Yaskawa INFORM job: X2_8B-21B(90,180)_DOD_WZMOC_BOK.JBI

/JOB
//NAME X2_8B-21B(90,180)_DOD_WZMOC_BOK
///FOLDERNAME X2
//POS
///NPOS 1035,1035,1035,44,0,0
///TOOL 0
///POSTYPE PULSE
///PULSE
C00000=-1415,-134459,-133802,-1969,12985,79332
C00001=-87080,-112473,-103627,-41798,51237,70410
C00002=-91681,-107347,-99471,-39221,49165,68848
C00003=-93439,-105106,-97054,-38371,48113,68361
C00004=-93441,-104864,-95967,-38672,47682,68565
C00005=-93504,-104969,-96260,-38564,47753,68495
C00006=-95585,-102642,-95415,-36914,47385,67494
C00007=-93504,-104969,-96260,-38564,47753,68495
C00008=-87147,-112175,-102116,-42180,50619,70689
C00009=-87145,-119394,-106475,-25944,48524,38750
C00010=-91166,-110510,-101811,-22693,48895,36705
C00011=-92650,-107060,-99920,-21494,49065,35962
C00012=-94767,-104655,-99060,-19829,49198,34943
C00013=-94484,-105085,-99259,-20052,49173,35080
C00014=-93721,-102513,-96995,-20598,49294,35408
C00015=-94484,-105085,-99259,-20052,49173,35080
C00016=-89209,-117497,-105909,-24366,48468,37757
C00017=-93166,-113214,-115710,-1969,57926,79332
C00018=-93710,-106990,-108704,-1652,56802,79139
C00019=-93766,-106412,-107148,-1629,56140,79127
C00020=-93768,-106433,-106329,-1638,55626,79135
C00021=-93918,-105383,-106173,-1535,56065,79069
C00022=-94164,-101296,-104676,-1361,57240,78956
C00023=-93895,-105502,-106499,-1547,56205,79076
C00024=-93151,-113316,-114305,-1998,57010,79354
C00025=-81072,-99391,-111155,-4750,63110,78553
C00026=-81984,-95120,-104767,-4287,61328,78293
C00027=-82103,-94682,-103397,-4241,60705,78273
C00028=-82106,-94924,-102383,-4271,59960,78300
C00029=-82089,-94934,-102578,-4276,60076,78302
C00030=-82803,-90374,-100753,-3806,61258,77993
C00031=-82089,-94934,-102578,-4276,60076,78302
C00032=-81057,-100006,-109908,-4804,62030,78604
C00033=-94004,-119945,-107122,49530,42714,48164
C00034=-93972,-116281,-97047,53343,39935,45878
C00035=-92833,-103149,-88492,51302,40218,47068
C00036=-93174,-100930,-87132,51219,40604,47120
C00037=-93174,-100493,-85792,51770,40220,46795
C00038=-93174,-101015,-87399,51095,40684,47186
C00039=-92955,-97894,-86230,50180,41136,47726
C00040=-93303,-100448,-87190,51023,40860,47230
C00041=-98055,-98607,-86499,53149,43882,46024
C00042=-96642,-96320,-85623,51883,43475,46780
C00043=-95342,-96864,-85830,51299,42647,47109
C00044=-97130,-98187,-86063,52744,43317,46271
C00045=-114545,-105110,-100746,39625,57097,48369
C00046=-113947,-102413,-97570,39574,56382,48359
C00047=-113947,-102278,-96691,39772,56015,48196
C00048=-113346,-99976,-96570,39024,56612,48763
C00049=-112899,-98120,-95866,38597,56823,49078
C00050=-114020,-99555,-96940,39169,57262,48705
C00051=-56302,-84822,-83054,-58022,66572,84014
C00052=-58361,-85953,-83540,-57558,65172,83717
C00053=-56302,-84822,-83054,-58022,66572,84014
C00054=-50122,-85714,-86741,-59061,71306,84454
C00055=-54195,-101901,-111197,-24063,62262,77343
C00056=-67243,-111926,-101536,21450,29925,69540
C00057=-66442,-101704,-94400,19916,30532,70304
C00058=-66308,-99858,-92576,19846,30336,70336
C00059=-66311,-99589,-91307,20230,29731,70137
C00060=-66308,-99960,-93112,19687,30597,70418
C00061=-70591,-100617,-92786,25268,31264,67678
C00062=-70591,-100325,-91437,25755,30647,67424
C00063=-68222,-99738,-91214,22742,30105,68906
C00064=-70591,-100606,-92729,25289,31242,67667
C00065=-66097,-110297,-96199,21577,27345,69446
C00066=-65719,-107666,-92844,21562,26575,69447
C00067=-65848,-106528,-92445,21497,26927,69482
C00068=-65365,-110699,-93884,21743,25627,69354
C00069=-67243,-111926,-101536,21450,29925,69540
C00070=-68963,-41843,-96211,-398,96948,-48811
C00071=-76932,-51697,-92360,2602,89609,-51106
C00072=-71886,-45093,-85416,705,88639,-49643
C00073=-71886,-45937,-84760,705,87803,-49648
C00074=-71886,-44632,-85753,705,89084,-49641
C00075=-68776,-90352,-95136,-4313,51281,-47645
C00076=-68803,-86754,-93636,-4241,52203,-47695
C00077=-68762,-92243,-95906,-4353,50785,-47617
C00078=-77446,-64871,-91176,8832,74282,-49527
C00079=-75907,-64612,-91046,8095,74185,-49034
C00080=-78150,-64967,-91224,9168,74335,-49752
C00081=-78150,-57569,-97635,8943,81990,-49191
C00082=-68963,-41843,-96211,-398,96948,-48811
C00083=-67385,-42511,-92598,-992,94393,-48367
C00084=-66773,-44328,-90253,-1220,92024,-48175
C00085=-66900,-44765,-89647,-1171,91425,-48205
C00086=-66773,-43962,-90441,-1221,92327,-48178
C00087=-69817,-49291,-93527,-72,91467,-49038
C00088=-102407,-61387,-79216,48101,75803,-74984
C00089=-99741,-62884,-79905,47237,74215,-74494
C00090=-102407,-61387,-79216,48101,75803,-74984
C00091=-71396,-101707,-96198,105,39560,-49678
C00092=-71544,-99303,-95354,247,40276,-49753
C00093=-71126,-105930,-97636,-165,38275,-49535
C00094=-74447,-120283,-111838,3099,39699,-51260
C00095=-57750,-84762,-113304,-22338,79933,-80646
C00096=-38298,-117376,-123136,-35520,84192,-83183
C00097=-31003,-114098,-105660,-45955,85390,-81321
C00098=-32496,-116782,-107403,-45795,84408,-81579
C00099=-34116,-118987,-108120,-45640,83088,-81742
C00100=-33779,-118873,-108083,-45678,83285,-81673
C00101=-33779,-118389,-106291,-45736,82677,-81394
C00102=-33116,-116007,-107005,-45711,84199,-81779
C00103=-43122,-77390,-91933,-43525,86904,-87571
C00104=-44353,-78017,-92219,-43231,86215,-87819
C00105=-45440,-79271,-92786,-42975,85486,-87990
C00106=-45102,-79332,-92813,-43057,85636,-87902
C00107=-45102,-79709,-91490,-43095,84888,-87585
C00108=-41853,-68825,-87871,-43817,88900,-87868
C00109=-48095,-31712,-66541,-47290,99218,-86920
C00110=-48762,-33638,-67810,-47108,98755,-86994
C00111=-49503,-35735,-69173,-46902,98237,-87073
C00112=-49389,-35416,-68966,-46933,98317,-87062
C00113=-49389,-36060,-68028,-46814,97684,-86756
C00114=-48487,-32850,-67294,-47182,98948,-86964
C00115=-45126,-25671,-76382,-49967,106798,-89554
C00116=-48508,-32956,-85951,-38791,109748,-85822
C00117=-73491,-115415,-129730,-12591,84406,-82629
C00118=-68604,-111632,-124361,34026,103601,-55041
C00119=-52690,-105642,-114364,31889,95098,-51390
C00120=-50963,-109289,-114635,31553,93010,-51314
C00121=-50968,-109442,-114037,31534,92627,-51422
C00122=-50963,-109237,-114816,31559,93129,-51281
C00123=-54701,-101748,-112541,32228,96580,-51739
C00124=-54580,-102143,-110625,32107,95358,-52042
C00125=-52710,-105778,-111943,31798,93771,-51772
C00126=-54580,-102143,-110625,32107,95358,-52042
C00127=-53574,-106836,-112314,31893,93817,-52092
C00128=-52008,-102475,-110737,31756,94333,-51344
C00129=-53574,-106836,-112314,31893,93817,-52092
C00130=-61074,-96775,-114868,33501,102293,-52496
C00131=-149084,-102156,-129577,22032,95315,-42360
C00132=-128569,-114069,-129208,14930,94899,-36248
C00133=-124702,-111484,-125119,14131,93099,-35189
C00134=-123206,-111006,-122572,13804,91571,-34868
C00135=-123205,-111346,-122108,13798,91123,-34918
C00136=-123169,-110975,-122344,13795,91444,-34870
C00137=-122647,-104244,-120003,13724,93323,-34489
C00138=-123169,-110975,-122344,13795,91444,-34870
C00139=-116503,-109521,-121739,12400,90787,-32743
C00140=-113941,-110266,-121994,11839,90202,-31960
C00141=-116503,-109521,-121739,12400,90787,-32743
C00142=-121595,-114825,-128025,13496,92670,-34216
C00143=-123984,-121300,-124584,22039,85383,-28695
C00144=-118596,-113071,-118409,20758,84424,-26972
C00145=-117828,-112575,-117002,20585,83663,-26833
C00146=-117596,-112721,-116348,20543,83158,-26838
C00147=-117643,-112201,-116474,20543,83493,-26797
C00148=-117846,-106122,-114344,20549,85245,-26570
C00149=-117643,-112201,-116474,20543,83493,-26797
C00150=-125192,-113488,-115877,22341,84450,-29296
C00151=-124919,-116220,-115928,22323,83104,-29449
C00152=-122352,-116155,-116251,21738,82647,-28614
C00153=-124919,-116220,-115928,22323,83104,-29449
C00154=-123984,-121300,-124584,22039,85383,-28695
C00155=-86442,-134681,-133724,-19248,79211,-32552
C00156=-86002,-121949,-124889,-19319,80358,-32581
C00157=-85994,-121959,-123892,-19351,79775,-32484
C00158=-85995,-122137,-123177,-19379,79272,-32404
C00159=-85938,-122450,-123568,-19392,79360,-32398
C00160=-86651,-115539,-121342,-19081,81262,-32951
C00161=-85938,-122450,-123568,-19392,79360,-32398
C00162=-130270,-119263,-121891,15868,79169,-48216
C00163=-132135,-133974,-122544,16883,72658,-49767
C00164=-129371,-136174,-123179,16117,71390,-48932
C00165=-132135,-133974,-122544,16883,72658,-49767
C00166=-120611,-122953,-119681,21560,80854,-22535
C00167=-120610,-122943,-118608,21593,80243,-22645
C00168=-120610,-122853,-116921,21650,79318,-22813
C00169=-120610,-122881,-117271,21638,79506,-22779
C00170=-120610,-122878,-117279,21638,79511,-22778
C00171=-120610,-122881,-117271,21638,79506,-22779
C00172=-120610,-122873,-117198,21640,79468,-22785
C00173=-120610,-122853,-117190,21640,79473,-22785
C00174=-120610,-122873,-117198,21640,79468,-22785
C00175=-120611,-122910,-120952,21522,81605,-22399
C00176=-86002,-120340,-127953,-19212,82925,-32989
C00177=-85994,-121959,-123892,-19351,79775,-32484
C00178=-85995,-122137,-123177,-19379,79272,-32404
C00179=-85938,-122450,-123568,-19392,79360,-32398
C00180=-86651,-115539,-121342,-19081,81262,-32951
C00181=-85938,-122450,-123568,-19392,79360,-32398
C00182=-130270,-119263,-121891,15868,79169,-48216
C00183=-132135,-133974,-122544,16883,72658,-49767
C00184=-129371,-136174,-123179,16117,71390,-48932
C00185=-132135,-133974,-122544,16883,72658,-49767
C00186=-120612,-120891,-127143,3106,87300,-4415
C00187=-120611,-122177,-124352,3111,84925,-4474
C00188=-120611,-122645,-122467,3116,83527,-4507
C00189=-120611,-122779,-121606,3119,82929,-4523
C00190=-120611,-122697,-122159,3117,83311,-4513
C00191=-120611,-122692,-122166,3117,83318,-4513
C00192=-120611,-122697,-122159,3117,83311,-4513
C00193=-120611,-121412,-126223,3107,86468,-4436
C00194=-96873,-135896,-136150,20148,98342,-27274
C00195=-53188,-122774,-119059,34227,101931,-42117
C00196=-53187,-122644,-116623,34032,100735,-42492
C00197=-53184,-122447,-115007,33919,99986,-42724
C00198=-53180,-122268,-113886,33849,99484,-42877
C00199=-53186,-122531,-115629,33961,100272,-42636
C00200=-53233,-122033,-113114,32057,113501,-44659
C00201=-53229,-122037,-113108,32057,113495,-44659
C00202=-53233,-122033,-113114,32057,113501,-44659
C00203=-53127,-122157,-112856,34567,84618,-41563
C00204=-53132,-122146,-112848,34568,84621,-41564
C00205=-53127,-122157,-112856,34567,84618,-41563
C00206=-53124,-122720,-116247,34514,86111,-41098
C00207=-61684,-126457,-131749,21672,103686,-55019
C00208=-68676,-133744,-131015,10578,108811,-68614
C00209=-80160,-118182,-130261,-41,125141,-81817
C00210=-80187,-122370,-123619,-70,118933,-81856
C00211=-80183,-122639,-122398,-68,118043,-81854
C00212=-80181,-122756,-121636,-67,117515,-81853
C00213=-80184,-122603,-122588,-68,118179,-81854
C00214=-80182,-122615,-122584,-67,118170,-81853
C00215=-80184,-122603,-122588,-68,118179,-81854
C00216=-80200,-121154,-126606,-75,121396,-81862
C00217=-109164,-117358,-132635,-7350,119146,-48306
C00218=-144183,-119511,-130571,-15498,107286,-7245
C00219=-197934,-122815,-127402,-28006,89082,55776
C00220=-202772,-123889,-124791,-27048,85608,54814
C00221=-204705,-124106,-122314,-26692,83530,54575
C00222=-204705,-124189,-120905,-26732,82711,54762
C00223=-205113,-122699,-120601,-26621,83104,54520
C00224=-208506,-122040,-120392,-25870,82241,53457
C00225=-204510,-125657,-121990,-26775,82699,54838
C00226=-204510,-125393,-124777,-26704,84359,54459
C00227=-217123,-144581,-130617,-26990,80795,43719
C00228=-208514,-157553,-136215,-22784,79668,13108
C00229=-208134,-153606,-128050,-23049,77001,13769
C00230=-209226,-147410,-126429,-22728,78719,13024
C00231=-208514,-151468,-127497,-22936,77598,13510
C00232=-208514,-156517,-134755,-22805,79329,13174
C00233=-197934,-122815,-127402,-28006,89082,55776
C00234=-202772,-123889,-124791,-27048,85608,54814
C00235=-204705,-124106,-122314,-26692,83530,54575
C00236=-204705,-124189,-120905,-26732,82711,54762
C00237=-205113,-122699,-120601,-26621,83104,54520
C00238=-208506,-122040,-120392,-25870,82241,53457
C00239=-204510,-125657,-121990,-26775,82699,54838
C00240=-204510,-125393,-124777,-26704,84359,54459
C00241=-217123,-144581,-130617,-26990,80795,43719
C00242=-217745,-144568,-135920,-20596,85340,27526
C00243=-208514,-151468,-127497,-22936,77598,13510
C00244=-209226,-147410,-126429,-22728,78719,13024
C00245=-208514,-151468,-127497,-22936,77598,13510
C00246=-208514,-156517,-134755,-22805,79329,13174
C00247=-187736,-116553,-120968,-36188,98329,31010
C00248=-144869,-104708,-130913,697,92502,-12445
C00249=-97478,-100538,-119508,25976,122096,-72949
C00250=-94415,-115583,-120723,24602,114867,-73486
C00251=-94145,-116737,-119872,24403,113768,-73630
C00252=-94090,-116915,-118863,24267,113100,-73760
C00253=-94227,-118887,-121662,24392,113788,-73658
C00254=-94618,-126072,-123928,23885,111795,-74261
C00255=-93811,-121058,-122280,24303,112998,-73673
C00256=-123165,-134656,-120887,30393,109989,-65140
C00257=-122877,-135920,-118822,30065,108215,-65520
C00258=-120918,-135771,-118381,30417,107339,-64954
C00259=-122877,-135920,-118822,30065,108215,-65520
C00260=-123434,-129548,-123417,31323,113703,-64157
C00261=-126606,-101457,-128935,16844,101795,-36174
C00262=-152779,-135138,-131563,2515,76140,-19155
C00263=-150820,-122490,-124749,1875,78392,-18455
C00264=-150097,-118368,-121531,1645,78513,-18212
C00265=-150095,-118599,-120646,1648,77850,-18220
C00266=-147666,-112236,-119185,871,80184,-17389
C00267=-146670,-110099,-118456,556,80825,-17059
C00268=-148658,-114325,-119887,1186,79554,-17722
C00269=-87079,-91764,-103818,-42328,107533,9448
C00270=-87027,-91004,-101788,-42122,106912,9740
C00271=-89264,-90509,-101588,-42089,105978,9119
C00272=-87027,-91004,-101788,-42122,106912,9740
C00273=-87391,-90282,-107909,-43186,109836,8282
C00274=-92115,-87061,-118989,-19004,94950,-3823
C00275=-78975,-130870,-123203,19746,71053,-12291
C00276=-74317,-97013,-111518,17407,83606,-9286
C00277=-74211,-95430,-110119,17377,83539,-9259
C00278=-74211,-95892,-109317,17397,82840,-9358
C00279=-75305,-113551,-114600,17838,69768,-10493
C00280=-78326,-111051,-111958,19079,70114,-11550
C00281=-78379,-106110,-110225,18937,71523,-11339
C00282=-78263,-116865,-113913,19272,68408,-11810
C00283=-85880,-113569,-112821,22054,71256,-14152
C00284=-85920,-114580,-110580,22309,69503,-14507
C00285=-82054,-114988,-110714,20879,68380,-13249
C00286=-85920,-114580,-110580,22309,69503,-14507
C00287=-78975,-130870,-123203,19746,67177,-12291
C00288=-159950,-115131,-126913,-23322,109234,64770
C00289=-163413,-124246,-126581,-22686,103792,64589
C00290=-164859,-127477,-125491,-22457,101245,64551
C00291=-164857,-127553,-124648,-22406,100728,64651
C00292=-164862,-127370,-126252,-22506,101730,64457
C00293=-158275,-145382,-129341,-21795,96649,67831
C00294=-159759,-153222,-131425,-21726,93697,67826
C00295=-158275,-145382,-129341,-21795,96649,67831
C00296=-157577,-144643,-126617,-21696,95625,68274
C00297=-160219,-140867,-125578,-21868,96138,67212
C00298=-157577,-144643,-126617,-21696,95625,68274
C00299=-152631,-134238,-128202,-21932,102817,68768
C00300=-146941,-123801,-133763,-3444,102850,52685
C00301=-136178,-116173,-124987,31736,84906,22811
C00302=-134413,-106132,-117362,31242,84680,23412
C00303=-134231,-105594,-115694,31219,83968,23286
C00304=-134230,-105863,-115134,31239,83552,23172
C00305=-134007,-104199,-114803,31151,84035,23389
C00306=-133473,-100630,-113499,30965,84737,23780
C00307=-134315,-106237,-115533,31260,83629,23161
C00308=-136272,-117460,-124003,31807,83855,22481
C00309=-136226,-116324,-125056,31750,84893,22789
C00310=-134474,-106353,-117504,31259,84679,23389
C00311=-134275,-105758,-115681,31235,83904,23252
C00312=-134274,-105987,-115198,31252,83547,23154
C00313=-134027,-104733,-115029,31162,83924,23350
C00314=-133465,-100971,-113658,30966,84667,23763
C00315=-134308,-106598,-115693,31262,83551,23142
C00316=-136269,-117902,-124178,31812,83752,22453
C00317=-139753,-124875,-130430,383,75663,-26245
C00318=-143223,-157944,-133481,-5653,58679,-38405
C00319=-140983,-144085,-126452,-6488,61628,-37698
C00320=-140148,-138933,-122655,-6835,62006,-37402
C00321=-140147,-138616,-121921,-6853,61719,-37384
C00322=-140691,-136506,-121897,-6553,62737,-37651
C00323=-138669,-131542,-120459,-7325,64564,-37004
C00324=-140691,-136506,-121897,-6553,62737,-37651
C00325=-145148,-139028,-124584,-4588,62787,-39337
C00326=-159973,-92454,-110285,14523,90938,-48717
C00327=-158765,-97223,-112137,14224,89465,-48492
C00328=-159973,-92454,-110285,14523,90938,-48717
C00329=-164681,-91509,-114703,15696,94847,-49769
C00330=-142525,-105883,-132766,-7713,103357,-60336
C00331=-90751,-115691,-121566,-36045,104861,-61043
C00332=-92920,-122587,-117773,-35137,99152,-60047
C00333=-93124,-123070,-117553,-35091,98753,-60003
C00334=-93124,-123008,-116878,-35050,98435,-59900
C00335=-93160,-123063,-117190,-35068,98555,-59953
C00336=-95752,-125144,-117838,-34977,96947,-60505
C00337=-93160,-123063,-117190,-35068,98555,-59953
C00338=-92038,-109836,-114685,-38536,89453,-57060
C00339=-86810,-100893,-104585,-47463,92019,-56975
C00340=-88449,-102594,-103600,-47188,90148,-56855
C00341=-88449,-102618,-102426,-47172,89639,-56610
C00342=-88449,-102603,-103366,-47184,90046,-56806
C00343=-85133,-99388,-102162,-47637,92393,-56350
C00344=-85168,-99488,-101153,-47595,91912,-56132
C00345=-86978,-101259,-101820,-47360,90627,-56378
C00346=-84037,-98201,-102123,-47804,93363,-56297
C00347=-108771,-112096,-123986,-16313,85813,-59347
C00348=-109769,-112695,-132242,-3132,99947,-61138
C00349=-127404,-127157,-120795,27540,73197,-60883
C00350=-120526,-123085,-115007,25540,69700,-59025
C00351=-119461,-122312,-114032,25210,69192,-58723
C00352=-119461,-122116,-113003,25293,68708,-58832
C00353=-119461,-122312,-114032,25210,69192,-58723
C00354=-94655,-112249,-115827,-1041,75214,-51009
C00355=-93364,-111129,-115444,-1499,75574,-50577
C00356=-121213,-123445,-114215,25873,69302,-59387
C00357=-127714,-127278,-119628,27738,72603,-61150
C00358=-140848,-129628,-128054,17424,84805,-27418
C00359=-127903,-106251,-120637,17388,91568,-15860
C00360=-124887,-98361,-114445,16717,91208,-14907
C00361=-124614,-94849,-112077,16660,91489,-14780
C00362=-117832,-103976,-115449,15062,87719,-13014
C00363=-118209,-109888,-118953,15141,86934,-13233
C00364=-120968,-118649,-124805,15800,86569,-14208
C00365=-112726,-101228,-128594,1890,90279,15897
C00366=-102865,-105549,-130121,-1361,88970,18873
C00367=-85416,-143080,-122146,-23399,58401,32529
C00368=-89847,-131888,-116792,-20882,59491,30436
C00369=-92125,-126361,-114096,-19602,60042,29398
C00370=-92108,-126361,-114086,-19611,60041,29405
C00371=-94963,-119193,-112807,-13876,65309,25883
C00372=-99230,-109273,-111594,-7832,72910,21884
C00373=-97558,-114678,-114533,-8498,72116,22521
C00374=-94805,-124749,-120489,-9597,70928,23580
C00375=-89899,-115674,-129227,-15589,81503,27304
C00376=-94000,-113154,-130859,1035,116659,-75004
C00377=-93721,-118000,-129934,5060,122177,-74127
C00378=-93715,-120352,-127357,4900,119392,-74256
C00379=-95346,-120435,-125547,4467,118331,-74923
C00380=-87734,-123112,-126247,6115,116903,-72103
C00381=-93725,-120284,-127319,4898,119404,-74259
C00382=-93731,-117931,-129895,5059,122189,-74130
C00383=-92605,-107385,-114202,-42080,118626,-78084
C00384=-94957,-117308,-114744,-40643,113912,-77125
C00385=-96859,-119647,-113709,-40343,111617,-77062
C00386=-96820,-119688,-113698,-40330,111613,-77042
C00387=-92369,-120637,-111842,-39132,112371,-75247
C00388=-87506,-133441,-114197,-38673,106213,-75021
C00389=-90618,-118755,-112828,-39302,114392,-75239
C00390=-88476,-109244,-112462,-40625,118981,-76164
C00391=-73726,-95231,-122050,-23824,117115,-78775
C00392=-68964,-113071,-130294,19412,109419,-80322
C00393=-55630,-112625,-122011,35520,97927,-81697
C00394=-52390,-118820,-120628,34805,93310,-81881
C00395=-47869,-106069,-116317,31727,98681,-78960
C00396=-58944,-112669,-113031,37596,97582,-82877
C00397=-56690,-122472,-119439,35129,92879,-83747
C00398=-59872,-116629,-120975,35716,97415,-83571
C00399=-61517,-148095,-119735,48293,75564,-80066
C00400=-55473,-148057,-116974,48060,71191,-79214
C00401=-53771,-146175,-114985,47935,70110,-78894
C00402=-54494,-144748,-112549,48210,69974,-79344
C00403=-55476,-147094,-115701,48129,70996,-79318
C00404=-61520,-147186,-118480,48348,75358,-80173
C00405=-87978,-108563,-128727,6750,125872,-71649
C00406=-93715,-120352,-127357,4900,119392,-74256
C00407=-94869,-122678,-126412,4545,117687,-74766
C00408=-87426,-125031,-126928,6148,116319,-72021
C00409=-93725,-120284,-127319,4898,119404,-74259
C00410=-93731,-117931,-129895,5059,122189,-74130
C00411=-92605,-107385,-114202,-42080,118626,-78084
C00412=-94957,-117308,-114744,-40643,113912,-77125
C00413=-96631,-121222,-114212,-40163,111336,-76837
C00414=-96582,-121324,-114222,-40145,111323,-76807
C00415=-92276,-122277,-112363,-38961,112002,-75057
C00416=-87192,-135738,-114687,-38435,105658,-74669
C00417=-90618,-118755,-112828,-39302,114392,-75239
C00418=-88476,-109244,-112462,-40625,118981,-76164
C00419=-73726,-95231,-122050,-23824,117115,-78775
C00420=-68964,-113071,-130294,19412,109419,-80322
C00421=-55630,-112625,-122011,35520,97927,-81697
C00422=-52390,-118820,-120628,34805,93310,-81881
C00423=-47557,-106620,-116510,31676,98430,-78912
C00424=-58659,-113116,-113184,37566,97351,-82838
C00425=-56690,-122472,-119439,35129,92879,-83747
C00426=-59872,-116629,-120975,35716,97415,-83571
C00427=-61517,-148095,-119735,48293,75564,-80066
C00428=-55473,-148057,-116974,48060,71191,-79214
C00429=-53043,-147267,-115261,47953,69457,-78858
C00430=-53748,-146178,-113424,48182,69442,-79233
C00431=-55476,-147094,-115701,48129,70996,-79318
C00432=-61520,-147186,-118480,48348,75358,-80173
C00433=-69196,-132761,-125763,48066,87564,-77891
C00434=-67178,-112107,-133350,-9560,121946,-71499
C00435=-53652,-115588,-130730,-10921,119132,-80041
C00436=-53631,-118653,-128170,-10572,116038,-79726
C00437=-49406,-129162,-130962,-9295,109096,-77614
C00438=-56866,-119557,-126808,-10903,114346,-80761
C00439=-54665,-117852,-125979,-10629,114989,-80007
C00440=-57520,-119011,-127190,-3009,114777,-80027
C00441=-59278,-121853,-127991,842,113579,-80159
C00442=-55695,-120300,-124998,1328,112531,-78914
C00443=-53493,-120154,-126714,1639,113579,-78070
C00444=-53512,-117734,-129516,1682,116546,-78033
C00445=-64263,-112177,-127274,18013,116425,-52133
C00446=-53349,-113292,-116223,34708,105130,-41711
C00447=-53347,-113647,-113946,34435,103813,-42137
C00448=-52680,-112871,-112467,34368,103124,-42082
C00449=-58031,-122280,-112065,36284,98076,-45699
C00450=-53343,-113729,-112902,34324,103242,-42318
C00451=-53345,-113489,-115217,34581,104530,-41905
C00452=-83368,-135406,-127982,43757,111124,24122
C00453=-107112,-148704,-121184,48737,110155,73723
C00454=-107085,-142005,-111593,48000,108472,72828
C00455=-107084,-140010,-108705,47787,107957,72557
C00456=-87331,-137626,-115833,38185,104318,80918
C00457=-107143,-152743,-127540,-1092,113262,57657
C00458=-106498,-152435,-127519,-1673,113318,57021
C00459=-107059,-148801,-134211,-1989,119286,56706
C00460=-109333,-147161,-118098,47834,110594,72761
C00461=-109333,-141938,-110765,47268,109335,72096
C00462=-106839,-147244,-109723,47050,105697,71521
C00463=-96955,-158208,-128899,-2670,111185,56030
C00464=-107130,-144670,-115956,-40497,90070,47196
C00465=-107133,-145289,-116877,-40503,90261,47122
C00466=-107139,-146938,-119316,-40521,90762,46927
C00467=-81304,-146505,-131302,-46256,99624,33732
C00468=-42290,-135810,-134986,-6789,56953,-43412
C00469=-53482,-111499,-99357,-5283,31563,-44884
C00470=-53488,-110753,-96932,-5448,30458,-44798
C00471=-53106,-110845,-96482,-5998,30161,-44520
C00472=-53143,-110117,-93832,-6189,28906,-44421
C00473=-53188,-109818,-93168,-6175,28651,-44427
C00474=-53095,-108922,-90553,-6542,27518,-44240
C00475=-53472,-108968,-91791,-5862,28222,-44586
C00476=-53466,-109889,-94290,-5675,29282,-44681
C00477=-93748,-113667,-111432,27227,62688,-41579
C00478=-93751,-113561,-109328,27520,61581,-41869
C00479=-94535,-110348,-107800,27711,62471,-41963
C00480=-94560,-109570,-102150,28499,59749,-42715
C00481=-93743,-112935,-104615,28181,59286,-42489
C00482=-93741,-113330,-106821,27872,60309,-42206
C00483=-53707,-103235,-126817,-3349,90409,-72793
C00484=-53694,-107630,-124107,-3352,86490,-72685
C00485=-53689,-108955,-122884,-3357,85060,-72645
C00486=-53697,-108940,-122873,-3354,85062,-72648
C00487=-53721,-108898,-122839,-3346,85062,-72656
C00488=-53729,-108884,-122827,-3345,85059,-72658
C00489=-53735,-107561,-124050,-3339,86489,-72698
C00490=-53748,-103173,-126762,-3336,90406,-72805
C00491=-44251,-68518,-112793,-6305,100072,-70363
C00492=-80270,30794,-42629,-11133,115571,-76543
C00493=-69737,67118,16632,-42575,112328,-80617
C00494=-69636,63823,22197,-49512,110599,-81416
C00495=-67564,55530,12856,-50142,112647,-81508
C00496=-66424,44944,1253,-49852,108764,-84350
C00497=-65618,29495,-14632,-48008,102670,-88237
C00498=-64581,15750,-27557,-48396,103780,-88326
C00499=-64160,11595,-31362,-48525,104124,-88308
C00500=-61878,-10748,-50140,-48981,105285,-87846
C00501=-62672,195,-41330,-51307,112408,-84907
C00502=-58944,10301,-35991,-52571,115494,-84879
C00503=-69716,-6230,-69222,-29298,97742,-75748
C00504=-102330,-22799,-82036,11222,88832,-73278
C00505=-48313,-118911,-129560,19207,92704,-27073
C00506=-53495,-110604,-121584,20154,93282,-28749
C00507=-53898,-112894,-120750,20179,91787,-29140
C00508=-54091,-109968,-119805,20238,92698,-29053
C00509=-54227,-109896,-119946,20266,92849,-29073
C00510=-54259,-112639,-122766,20278,93161,-29031
C00511=-53522,-108468,-123882,20258,95652,-28360
C00512=-66910,-101677,-117691,1645,82254,17515
C00513=-66905,-103395,-115374,1652,79946,17486
C00514=-66559,-103374,-114061,1536,79140,17588
C00515=-66525,-103141,-114029,1523,79241,17602
C00516=-67620,-103650,-114144,1902,79074,17240
C00517=-69811,-106122,-108316,12679,69437,17327
C00518=-66783,-105788,-110032,11324,70201,18483
C00519=-66785,-105108,-112553,11207,72068,18659
C00520=-34610,-119076,-126707,-31995,89279,47352
C00521=-26693,-119602,-105841,-51320,82883,62074
C00522=-26676,-118953,-103885,-51392,82336,62389
C00523=-26611,-118260,-103653,-51381,82509,62328
C00524=-26639,-116853,-99731,-51529,81413,62927
C00525=-26666,-118021,-101324,-51491,81640,62785
C00526=-26683,-118745,-103309,-51412,82173,62476
C00527=-26741,-121947,-116429,-51038,86269,60171
C00528=-80158,-111738,-121779,-46707,81282,-33331
C00529=-80124,-114295,-114082,-47454,77096,-31277
C00530=-80115,-114367,-110881,-47781,75720,-30584
C00531=-79863,-115197,-109969,-48014,75178,-30182
C00532=-79793,-115451,-110067,-48044,75166,-30141
C00533=-80052,-114603,-110983,-47806,75713,-30548
C00534=-80061,-114542,-114188,-47480,77086,-31241
C00535=-80063,-113108,-120040,-30435,104055,-77976
C00536=-80050,-114212,-116860,-30086,101864,-77373
C00537=-80380,-112077,-114717,-30053,101557,-77419
C00538=-79932,-114590,-112006,-35005,85347,-77215
C00539=-79912,-114566,-112044,-35008,85386,-77219
C00540=-80479,-112475,-109427,-36632,80098,-77307
C00541=-80029,-114714,-111597,-36713,80437,-77233
C00542=-82440,-93132,-104306,-35744,84828,-79668
C00543=-83378,-90315,-100640,-35536,83784,-79702
C00544=-86724,-76310,-94495,-34501,85296,-81493
C00545=-81341,-82881,-101909,-35963,88366,-80388
C00546=-80042,-114535,-115070,-36542,82240,-77847
C00547=-80040,-111621,-122742,-8414,85267,-41918
C00548=-80035,-113457,-119567,-8450,82400,-41723
C00549=-81798,-124774,-120168,-7328,73182,-41674
C00550=-80327,-109577,-118133,2572,87034,-53415
C00551=-79380,-112621,-119090,2349,86031,-53125
C00552=-78889,-114029,-118891,6085,83597,-58153
C00553=-80002,-113603,-119620,10752,83390,-63441
C00554=-80006,-103113,-128729,10775,94202,-62513
C00555=-39776,-103787,-110683,-21075,62663,59255
C00556=-39766,-104399,-107995,-21452,60825,59622
C00557=-41663,-99518,-106576,-17765,63773,58656
C00558=-39441,-104963,-106701,-21848,59898,59942
C00559=-39326,-105104,-106740,-21922,59881,59993
C00560=-39744,-104425,-108009,-21464,60826,59630
C00561=-39754,-103814,-110697,-21087,62664,59263
C00562=-47977,-106691,-119962,-23629,83327,62671
C00563=-66867,-99660,-121232,-22132,99220,62132
C00564=-66851,-102572,-118810,-21937,96446,62653
C00565=-74494,-137000,-128982,-14609,78071,53501
C00566=-72467,-138184,-128020,-15181,77278,54315
C00567=-67516,-140688,-126942,-16493,76361,56201
C00568=-43056,-127353,-114280,-36292,85121,62743
C00569=-66851,-103895,-117201,-21852,94891,62938
C00570=-66868,-101493,-119792,-22004,97521,62449
C00571=-74321,-107832,-126985,11736,80239,61811
C00572=-66584,-114412,-108983,34198,49386,64476
C00573=-66581,-113854,-105403,35147,47795,63826
C00574=-59001,-125725,-103773,32485,32454,61113
C00575=-65790,-113886,-101008,36132,45231,63145
C00576=-65568,-123466,-98279,45853,34675,56822
C00577=-65581,-123771,-97752,46366,34344,56544
C00578=-66567,-113311,-102857,35821,46729,63375
C00579=-66569,-114089,-106515,34851,48256,64025
C00580=-52763,-107501,-118592,5184,62268,61653
C00581=-39766,-104399,-107995,-21452,60825,59622
C00582=-42284,-99628,-106389,-17466,63479,58468
C00583=-39837,-104496,-106407,-21621,59851,59791
C00584=-39825,-104515,-106407,-21630,59842,59799
C00585=-39744,-104425,-108009,-21464,60826,59630
C00586=-39754,-103814,-110697,-21087,62664,59263
C00587=-47977,-106691,-119962,-23629,83327,62671
C00588=-66867,-99660,-121232,-22132,99220,62132
C00589=-66851,-102572,-118810,-21937,96446,62653
C00590=-75086,-136456,-128394,-14464,77886,53317
C00591=-72467,-138185,-128020,-15181,77278,54315
C00592=-67516,-140689,-126942,-16493,76360,56201
C00593=-43574,-128187,-114530,-36250,84680,62675
C00594=-66851,-103895,-117201,-21852,94891,62938
C00595=-66868,-101493,-119792,-22004,97521,62449
C00596=-74321,-107832,-126985,11736,80239,61811
C00597=-66584,-114412,-108983,34198,49386,64476
C00598=-66581,-113854,-105403,35147,47795,63826
C00599=-59470,-125293,-103644,32823,32756,60929
C00600=-65940,-113573,-100903,36174,45372,63123
C00601=-65237,-123018,-98144,45460,34612,57042
C00602=-65306,-123403,-97643,46040,34287,56728
C00603=-66567,-113311,-102857,35821,46729,63375
C00604=-66569,-114089,-106515,34851,48256,64025
C00605=-66614,-114312,-115902,32344,53032,65825
C00606=-26293,-124733,-123676,35115,86081,77095
C00607=-26278,-124914,-120130,35186,84196,76502
C00608=-26550,-125631,-118910,35285,83385,76132
C00609=-26140,-123752,-118256,35186,83681,76394
C00610=-26301,-124893,-120124,35190,84211,76498
C00611=-26317,-124710,-123669,35119,86096,77090
C00612=-26368,-124828,-121889,39154,95960,78120
C00613=-26350,-124746,-118556,38992,94373,77544
C00614=-26342,-124553,-116950,38932,93670,77290
C00615=-26340,-123995,-113991,38847,92461,76851
C00616=-26347,-124286,-115407,38884,93032,77056
C00617=-26365,-124761,-118865,39006,94524,77592
C00618=-26264,-124528,-116402,47920,86072,68134
C00619=-26249,-123768,-112787,47988,84810,67516
C00620=-26243,-123374,-111311,48022,84325,67278
C00621=-26226,-122772,-109280,48074,83674,66962
C00622=-26232,-123227,-110778,48035,84146,67194
C00623=-26247,-124165,-114452,47952,85370,67795
C00624=-82585,-123093,-118421,52491,64599,59558
C00625=-107155,-118824,-102398,58122,50036,52281
C00626=-107155,-117467,-98958,59145,49269,51564
C00627=-96813,-117817,-104188,42223,47347,50994
C00628=-105933,-121077,-109912,10415,42869,62990
C00629=-105953,-121074,-109843,10442,42831,62975
C00630=-107149,-121400,-109798,11502,42801,62375
C00631=-106717,-121349,-105974,7567,38238,71665
C00632=-107169,-120346,-107141,7797,39493,71540
C00633=-108433,-119625,-117514,7930,46308,71537
C00634=-107111,-122100,-111275,39348,45202,56077
C00635=-107109,-117760,-98763,43179,41028,53713
C00636=-106761,-117495,-97713,43363,40478,53604
C00637=-106458,-119074,-102370,12274,36991,61895
C00638=-105683,-116022,-101280,9396,37560,63477
C00639=-85991,-103596,-98751,-25015,50891,70344
C00640=-83847,-106333,-107319,-25140,55050,70229
C00641=-110745,-121766,-106380,43469,44759,53583
C00642=-110745,-121766,-106380,43469,44759,53584
C00643=-120731,-110814,-96413,59684,53172,46713
C00644=-94986,-115649,-101302,-12294,38121,75258
C00645=-110957,-117259,-94521,-45268,37979,76630
C00646=-107127,-114270,-91297,-56630,43098,80056
C00647=-102543,-110504,-99650,-53136,49996,77723
C00648=-93612,-109275,-133010,12113,75674,64968
C00649=-74458,-81913,-116300,25886,107898,47202
C00650=-74285,-84923,-113224,25351,104735,46539
C00651=-74085,-86300,-112083,25142,103399,46313
C00652=-71499,-76504,-108067,25490,106819,45523
C00653=-62961,-60085,-100217,24652,107848,48688
C00654=-60437,-59805,-99888,23461,105440,51393
C00655=-60588,-58283,-100875,23679,106756,51616
C00656=-60637,-54628,-103477,24231,109960,52288
C00657=-76657,-70403,-83915,51355,64349,40407
C00658=-74830,-68241,-74355,53953,55282,38932
C00659=-73110,-62379,-68708,53436,54020,39148
C00660=-73126,-62440,-68450,53549,53912,39057
C00661=-36930,-67607,-75173,-26029,44061,77403
C00662=-80523,-89058,-85253,18218,36719,55154
C00663=-82272,-90569,-85112,18702,34759,56728
C00664=-81508,-95500,-88175,18158,33969,56993
C00665=-81043,-103588,-94156,17854,33413,57140
C00666=-82846,-88179,-88219,41798,48730,43563
C00667=-81818,-81213,-82326,41198,48211,43888
C00668=-79663,-80074,-80946,37957,46333,45127
C00669=-64011,-84834,-85332,4259,39755,58703
C00670=-75846,-87347,-86370,15921,40584,52659
C00671=-47572,-67654,-78731,-37306,60592,66422
C00672=-46339,-68382,-80235,-37741,61555,66618
C00673=-42699,-70655,-83815,-39176,63943,67342
C00674=-43803,-67144,-92021,-36183,69839,64523
C00675=-86906,-70734,-117845,25978,101850,24881
C00676=-194376,-118372,-116958,36622,58194,-75254
C00677=-187943,-106127,-101715,33777,52366,-74665
C00678=-187951,-105693,-98645,34509,50978,-75202
C00679=-187954,-105458,-97394,34809,50440,-75417
C00680=-187960,-105469,-97402,34805,50444,-75420
C00681=-187927,-105629,-98482,19599,46235,-60273
C00682=-187923,-105820,-99644,19403,46817,-60144
C00683=-187914,-106157,-102495,18928,48312,-59826
C00684=-188021,-109107,-91072,54887,40419,-77132
C00685=-188025,-108188,-88773,55807,39869,-77674
C00686=-188027,-107805,-87846,56180,39654,-77892
C00687=-188036,-107761,-87717,56242,39627,-77928
C00688=-188035,-108145,-88644,55869,39841,-77710
C00689=-188030,-109068,-90945,54948,40390,-77168
C00690=-188015,-114130,-110744,41340,72657,-75143
C00691=-188018,-113864,-107763,41683,71368,-75679
C00692=-188019,-113684,-106544,41824,70871,-75888
C00693=-188009,-113674,-106577,41816,70886,-75877
C00694=-188008,-113852,-107795,41674,71383,-75668
C00695=-188005,-114114,-110775,41332,72673,-75132
C00696=-187933,-113872,-110928,18210,58720,-57176
C00697=-187882,-113256,-105308,-719,43762,-42538
C00698=-187896,-112711,-102669,-725,42418,-42533
C00699=-187852,-113170,-101841,-775,41671,-42505
C00700=-187778,-112374,-98354,-1639,37547,-42296
C00701=-187899,-111729,-99017,-1491,38283,-42378
C00702=-187886,-112431,-101600,-1465,39511,-42393
C00703=-192869,-127835,-120494,22551,66263,-53872
C00704=-188079,-122619,-114609,40714,83609,-61664
C00705=-188077,-122103,-112045,40794,82601,-62056
C00706=-188097,-121812,-110726,41966,87288,-59780
C00707=-188097,-121769,-110559,41966,87227,-59806
C00708=-188105,-121282,-108770,41980,86589,-60067
C00709=-188106,-121566,-109755,41972,86936,-59927
C00710=-188110,-122188,-112187,41960,87826,-59570
C00711=-188058,-121965,-125191,40549,88870,-59628
C00712=-104402,-90439,-123637,22599,88102,26907
C00713=-80407,-121901,-119741,18448,66455,46046
C00714=-80400,-121844,-116068,18757,64334,45697
C00715=-80358,-121826,-114599,18875,63477,45568
C00716=-79500,-120626,-114191,18436,63629,45929
C00717=-80475,-121542,-115946,18779,64427,45684
C00718=-80482,-121578,-119613,18469,66554,46034
C00719=-85156,-144709,-129107,-21632,59402,64028
C00720=-93856,-120445,-109825,-39450,57641,70752
C00721=-93847,-119691,-106928,-40019,56559,71233
C00722=-86628,-99816,-98593,-45940,69277,74290
C00723=-86043,-99167,-98859,-45014,69635,74495
C00724=-83318,-93529,-94650,-47165,68336,75996
C00725=-93680,-116508,-100417,-40719,46210,72415
C00726=-93820,-118277,-102341,-40471,46353,72255
C00727=-93828,-119232,-105178,-39715,47322,71755
C00728=-93822,-120125,-107980,-28359,52237,38282
C00729=-93816,-119582,-106091,-28689,51458,38525
C00730=-93813,-119346,-105328,-28822,51152,38622
C00731=-93805,-118409,-102529,-29499,49391,39302
C00732=-93820,-119862,-107056,-29266,59584,40856
C00733=-93823,-120114,-107958,-29147,59957,40747
C00734=-93830,-120670,-110185,-28854,60909,40473
C00735=-63807,-119595,-131717,-32346,77391,31957
C00736=-66677,-121755,-125547,-9668,69981,-32239
C00737=-66675,-122709,-116301,-10101,63887,-31721
C00738=-66675,-122586,-115330,-10147,63360,-31673
C00739=-66678,-122782,-121307,9429,81851,-37654
C00740=-66765,-122962,-121469,9451,81867,-37681
C00741=-66675,-122328,-113778,33290,107246,-42961
C00742=-66675,-122499,-114776,33395,107690,-42822
C00743=-66677,-122795,-117228,33681,108831,-42458
C00744=-67830,-119002,-127241,35733,116022,-40496
C00745=-66677,-118144,-130351,-9432,74728,-32617
C00746=-66675,-122709,-116301,-10101,63887,-31721
C00747=-66675,-122566,-115195,-10154,63288,-31666
C00748=-66598,-122626,-121075,9408,81779,-37632
C00749=-62201,-135318,-124907,8438,77184,-36457
C00750=-72253,-125964,-118680,27296,92025,-49108
C00751=-76379,-123759,-128626,28058,99823,-48794
C00752=-71006,-123079,-126009,31798,108132,-44322
C00753=-66720,-122114,-124411,34847,112827,-41144
C00754=-125074,-112778,-121368,18538,134713,-61704
C00755=-173715,-145384,-131232,-10200,126221,-84589
C00756=-173715,-147046,-136936,-18176,117071,-78230
C00757=-173715,-145384,-131232,-55285,56270,-43989
C00758=-121435,-145384,-131232,-55285,56270,-43989
C00759=-118035,-115309,-97908,-59229,55500,-40903
C00760=-129283,-161545,-102403,-79044,40043,-30541
C00761=-116007,-110364,-98843,-57726,100679,-36272
C00762=-114757,-140924,-107985,-56048,95732,-32110
C00763=-114657,-138777,-101995,-58083,106215,-39512
C00764=-102008,-144788,-123359,-59173,119414,-41279
C00765=-15972,-110889,-128286,-10965,59905,-43045
C00766=-15972,-110889,-128286,-10965,59905,-43045
C00767=-101389,-60822,-75148,6919,68546,-70102
C00768=-115790,69230,64798,-8053,66131,-71909
C00769=-120688,105020,73307,-12402,84846,-73777
C00770=-120868,103639,75593,-12409,82749,-73629
C00771=-120940,103216,76680,-12418,81872,-73566
C00772=-120940,103732,79019,-12450,80724,-73451
C00773=-120940,103216,76680,-12418,81872,-73566
C00774=-120298,112004,89967,-12640,78393,-72988
C00775=-120707,106255,82361,-12511,80017,-73298
C00776=-120298,112004,89967,-12640,78393,-72988
C00777=-120228,112105,88453,-12614,79365,-73063
C00778=-120053,112844,85327,-12571,81642,-73235
C00779=-120830,71540,61874,-4756,55589,-66514
C00780=-120535,76858,72419,-5134,51864,-66212
C00781=-120418,79487,77321,-5314,50212,-66075
C00782=-120418,81305,81326,-5435,48689,-65991
C00783=-120418,79487,77321,-5314,50212,-66075
C00784=-121101,73566,71896,-4942,50464,-66384
C00785=-120640,77942,77238,-5256,49458,-66131
C00786=-121101,73566,71896,-4942,50464,-66384
C00787=-121222,71175,67349,-4775,52021,-66512
C00788=-121527,66226,57370,-4418,55590,-66797
C00789=-120817,46858,51705,6808,46216,-80289
C00790=-120487,52530,62238,7041,42645,-80409
C00791=-120357,55197,66992,7170,41090,-80474
C00792=-120357,57219,71131,7393,39594,-80606
C00793=-120357,55197,66992,7170,41090,-80474
C00794=-121171,51687,64922,7778,40638,-80922
C00795=-120657,55397,69123,7546,39918,-80729
C00796=-121171,51687,64922,7778,40638,-80922
C00797=-121307,49062,60252,7635,42163,-80850
C00798=-121648,43436,49847,7373,45678,-80715
C00799=-109578,66950,51259,-9202,73878,-70224
C00800=-101389,-60822,-75148,6919,68546,-70102
C00801=-96929,-90691,-89138,5080,61517,-23019
C00802=-96929,-90691,-89138,5080,61517,27168
C00803=-133997,38575,-5386,4879,105902,64390
C00804=-134430,35731,-4221,4855,103756,64161
C00805=-134605,34666,-3678,4847,102887,64068
C00806=-134604,34193,-2477,4825,101908,64030
C00807=-134605,34666,-3678,4847,102887,64068
C00808=-133324,38381,1851,4717,101326,64430
C00809=-133984,36157,-436,4773,101627,64224
C00810=-133324,38381,1851,4717,101326,64430
C00811=-132740,42105,45,4739,104308,64739
C00812=-159526,23962,790,32225,80504,55500
C00813=-158922,24925,5721,32299,78113,55050
C00814=-158682,25453,8443,32390,76826,54772
C00815=-158681,25549,9587,32465,76269,54609
C00816=-158682,25408,7790,32348,77149,54866
C00817=-160104,22984,7189,32780,76948,54233
C00818=-159169,24509,8648,32575,76492,54477
C00819=-160104,22984,7189,32780,76948,54233
C00820=-160967,21427,101,32642,80299,54873
C00821=-147551,27169,-6215,28445,81493,60312
C00822=-147017,27605,-1759,28452,79091,59917
C00823=-146805,27803,661,28506,77793,59674
C00824=-146803,27699,1600,28565,77235,59535
C00825=-146805,27874,109,28472,78126,59757
C00826=-148390,24338,-1607,29025,77984,59121
C00827=-147556,26192,183,28786,77573,59333
C00828=-148390,24338,-1607,29025,77984,59121
C00829=-149162,23542,-7999,28991,81344,59682
C00830=-129846,-17397,-52274,16165,101048,68229
C00831=-103949,-6271,-30701,7884,96105,76175
C00832=-94102,16895,-5866,4380,94047,79161
C00833=-94024,14878,-3719,4358,91692,79105
C00834=-93993,14152,-2780,4351,90742,79083
C00835=-93993,14253,-1030,4349,89719,79047
C00836=-93993,14152,-2780,4351,90742,79083
C00837=-93685,20015,4382,4321,89334,79138
C00838=-93881,17120,1686,4338,89515,79078
C00839=-93685,20015,4382,4321,89334,79138
C00840=-93796,22544,1176,4343,92603,79213
C00841=-95224,-25687,-42365,27028,60157,72238
C00842=-94111,-23276,-36997,26973,57954,72128
C00843=-93676,-22245,-34794,26967,57075,72081
C00844=-93677,-22196,-33100,27266,56165,71832
C00845=-93676,-22245,-34794,26967,57075,72081
C00846=-94165,-26445,-35973,27662,55954,71554
C00847=-93910,-23559,-33944,27450,56079,71704
C00848=-94165,-26445,-35973,27662,55954,71554
C00849=-95768,-30118,-43626,27714,58991,71694
C00850=-97625,-41604,-59467,17173,89706,-8843
C00851=-96114,-37688,-53918,16886,88057,-8555
C00852=-95526,-36022,-51615,16777,87400,-8443
C00853=-95527,-36150,-50037,16784,86406,-8579
C00854=-95526,-36022,-51615,16777,87400,-8443
C00855=-95532,-36183,-50637,16782,86745,-8534
C00856=-95234,-33170,-48668,16723,87008,-8396
C00857=-95532,-36183,-50637,16782,86745,-8534
C00858=-95504,-36095,-50208,16778,86530,-8554
C00859=-93996,-36675,-50581,16493,86163,-8084
C00860=-95504,-36095,-50208,16778,86530,-8554
C00861=-97625,-41604,-59467,17173,89706,-8843
C00862=-101873,-77751,-87156,42969,63075,62474
C00863=-95937,-74809,-81328,40948,58735,63434
C00864=-95565,-74583,-80935,40815,58468,63500
C00865=-95566,-74620,-79294,41227,57681,63141
C00866=-95565,-74583,-80935,40815,58468,63500
C00867=-98755,-73227,-80296,42221,60183,62682
C00868=-98803,-73638,-78797,42678,59356,62269
C00869=-96868,-74481,-79195,41849,58298,62761
C00870=-98803,-73638,-78797,42678,59356,62269
C00871=-97163,-69666,-76891,41573,59236,63045
C00872=-96752,-66139,-75134,41097,59602,63417
C00873=-97163,-69666,-76891,41573,59236,63045
C00874=-101873,-77751,-87156,42969,63075,62474
C00875=-126113,-49786,-51573,51544,90004,55144
C00876=-123973,-50127,-48217,51392,87374,54806
C00877=-123286,-49758,-46380,51349,86473,54664
C00878=-118478,-34750,-37348,50925,85086,56432
C00879=-119272,-35479,-39244,50973,86038,56539
C00880=-121232,-35158,-42579,51146,88553,56901
C00881=-111145,-57425,-62081,41633,61582,55088
C00882=-109620,-53993,-56645,41578,59663,54986
C00883=-109014,-52418,-54338,41560,58914,54950
C00884=-105531,-54881,-55720,40219,56972,55856
C00885=-106107,-56401,-57979,40230,57706,55889
C00886=-107578,-60042,-63488,40293,59558,55964
C00887=-93331,-25535,-46307,22677,87971,72102
C00888=-84242,-5399,-27465,11713,100257,81196
C00889=-83743,-8192,-25851,11599,97806,81134
C00890=-83603,-8644,-24372,11558,96668,81075
C00891=-80847,-8673,-24279,11462,96208,81977
C00892=-80973,-8366,-25985,11504,97411,82047
C00893=-81511,-5615,-27635,11617,99868,82095
C00894=-103949,-6271,-30701,7884,96105,76175
C00895=-129846,-17397,-52274,16165,101048,68229
C00896=-175693,57260,35469,48998,74273,48315
C00897=-174652,59964,42108,49342,71909,47593
C00898=-173987,58917,42535,48748,68669,47097
C00899=-173562,58305,42809,47399,62634,46211
C00900=-173482,53917,36869,46602,62532,46609
C00901=-174364,49990,29079,45939,64941,47387
C00902=-163099,39792,11105,47007,80916,54866
C00903=-161954,40669,15666,46993,78691,54338
C00904=-161675,41954,18470,47071,77805,54042
C00905=-160520,35916,12218,46685,77730,54566
C00906=-160850,34862,9687,46632,78611,54832
C00907=-162019,34035,5199,46665,80839,55343
C00908=-147988,42797,109,12455,106225,61454
C00909=-148219,40121,1423,12320,104123,61157
C00910=-148209,38525,1410,12269,103328,61081
C00911=-147238,35306,-1899,12234,103563,61431
C00912=-146513,33084,-4151,12206,103702,61693
C00913=-146794,35355,-3496,12271,104485,61677
C00914=-146567,38090,-4821,12411,106625,61976
C00915=-96929,-90691,-89138,5080,61517,27168
C00916=-96929,-90691,-89138,5080,61517,-23019
C00917=-101389,-60822,-75148,6919,68546,-70102
C00918=-109578,66950,51259,-9202,73878,-70224
C00919=-119285,73548,61078,-7759,54489,-67872
C00920=-119140,78931,71700,-8230,50768,-67516
C00921=-119083,81584,76629,-8462,49121,-67350
C00922=-122917,98444,98202,-6801,44189,-68705
C00923=-122308,90513,86215,-6785,47517,-68668
C00924=-122473,83260,72935,-6271,51921,-69036
C00925=-119074,82203,59752,-14757,75142,-72556
C00926=-112473,77653,55392,-16315,76732,-70397
C00927=-111583,66581,50085,-22599,68947,-68307
C00928=-112205,67748,51306,-22435,68636,-68485
C00929=-112291,70891,55012,-22505,67993,-68392
C00930=-120890,75924,58725,-8799,66214,-71114
C00931=-120891,72538,54662,-8752,66965,-71172
C00932=-121396,73617,55948,-8591,66676,-71337
C00933=-121396,72779,51526,-8459,68942,-71502
C00934=-134157,70152,49704,15847,72235,-43808
C00935=-133722,73949,59265,16087,68355,-44178
C00936=-133862,75249,62165,16247,67307,-44381
C00937=-129675,65866,51066,4701,64817,-31992
C00938=-128682,62362,47014,4314,65455,-31601
C00939=-130205,57581,36634,4742,69462,-32000
C00940=-130312,54578,33992,4779,69550,-32035
C00941=-129992,46081,35923,20239,67004,8502
C00942=-121496,43425,36833,5893,59088,22773
C00943=-120237,47252,43120,2387,56768,25932
C00944=-119972,47626,45454,2298,55515,26011
C00945=-128073,50557,47782,20949,62737,7811
C00946=-127834,53853,52717,21124,61417,7650
C00947=-123180,48310,46556,9691,56439,19302
C00948=-122651,35401,27095,8965,61652,19959
C00949=-109578,66950,51259,-9202,73878,-70224
C00950=-101389,-60822,-75148,6919,68546,-70102
C00951=-96929,-90691,-89138,5080,61517,-23019
C00952=-93242,-109726,-96296,3420,55961,28393
C00953=-92156,-22649,-39625,10516,94476,60392
C00954=-92549,-23820,-36378,10508,91967,60047
C00955=-92689,-24290,-35079,10509,90961,59915
C00956=-95254,-23373,-34430,10727,91365,59075
C00957=-94898,-22950,-35761,10710,92338,59280
C00958=-94492,-21797,-39017,10723,94837,59633
C00959=-92575,-26977,-42679,21088,73618,56030
C00960=-92430,-25186,-37423,21282,71416,55682
C00961=-92290,-24713,-35488,21345,70493,55566
C00962=-95616,-23226,-34216,23502,71566,54461
C00963=-95477,-23933,-36320,23344,72386,54682
C00964=-95719,-25683,-41558,23174,74597,55037
C00965=-96929,-90691,-89138,5080,61517,27168
C00966=-96929,-90691,-89138,5080,61517,-23019
C00967=-101389,-60822,-75148,6919,68546,-70102
C00968=-109578,66950,51259,-9202,73878,-70224
C00969=-108278,48890,46404,-6655,48460,-73563
C00970=-108252,54023,56228,-7048,45078,-73302
C00971=-108672,56895,61153,-6970,43500,-73378
C00972=-113114,65075,70630,-4174,41573,-75428
C00973=-112702,61866,65174,-4315,43297,-75310
C00974=-112766,56024,54314,-4011,46966,-75508
C00975=-103921,32533,46603,10708,30188,-75698
C00976=-104692,35200,60863,30413,16065,-83251
C00977=-104796,38679,66061,33302,14894,-84599
C00978=-102333,36267,63497,27606,14351,-81669
C00979=-100412,37194,55383,7603,26828,-73795
C00980=-100998,29868,43914,7479,30147,-73786
C00981=-109578,66950,51259,-9202,73878,-70224
C00982=-101389,-60822,-75148,6919,68546,-70102
C00983=-96929,-90691,-89138,5080,61517,-23019
C00984=-96929,-90691,-89138,5080,61517,27168
C00985=-90570,-23240,-39845,-1682,91658,61068
C00986=-90349,-1837,-19216,-4288,101242,62233
C00987=-90005,-3734,-19299,-4261,100340,62382
C00988=-92752,-2865,-18588,-4343,100202,61442
C00989=-95291,-22836,-35623,-1093,89189,59526
C00990=-94239,-22001,-38963,-1226,91687,59852
C00991=-90424,-29050,-43505,3763,58999,61302
C00992=-86008,-21130,-36360,-6353,62529,61992
C00993=-86454,-19207,-33152,-6175,61515,61881
C00994=-89453,-18520,-32647,-4592,61359,60761
C00995=-95351,-24457,-36663,6763,57473,59317
C00996=-94707,-27619,-42528,6252,59394,59681
C00997=-109011,-26713,-50438,8452,98222,74634
C00998=-144543,31549,-11380,-159,92982,60584
C00999=-143093,45679,4448,-4866,97184,60249
C01000=-143214,43522,5393,-4827,95492,60276
C01001=-146471,54490,17318,-4285,93619,59288
C01002=-148937,42537,3991,922,89189,59187
C01003=-148250,43318,770,754,91565,59420
C01004=-172279,3947,-14828,46151,77384,48319
C01005=-167570,-10636,-17777,41693,62852,42800
C01006=-166655,-7092,-11488,42082,60867,42363
C01007=-169056,5005,-1455,42887,62060,41693
C01008=-172859,17944,7820,47479,72977,45875
C01009=-174013,15583,1984,47261,75226,46421
C01010=-109011,-26713,-50438,8452,98222,74634
C01011=-99312,-50897,-61026,22837,72179,74454
C01012=-98138,-49989,-56545,22703,69739,74412
C01013=-106382,-52347,-50887,37007,65807,70627
C01014=-98813,-18962,-39289,22939,92751,75811
C01015=-101547,-27333,-44313,25543,91651,74875
C01016=-97857,-18198,-39852,20610,99055,76884
C01017=-96922,-25876,-47272,18742,95048,76352
C01018=-97638,-23312,-49453,18962,97729,76524
C01019=-81141,-50558,-66105,12803,46081,75388
C01020=-80687,-46119,-60183,12697,44679,75401
C01021=-80513,-44339,-57785,12667,44105,75401
C01022=-80516,-44488,-54802,13120,42239,75121
C01023=-80690,-46329,-57233,13145,42803,75122
C01024=-81145,-50923,-63237,13239,44177,75109
C01025=-83601,15534,-39616,9664,96262,77072
C01026=-80484,90945,50155,4324,118905,78550
C01027=-80490,84570,45509,4303,118490,78531
C01028=-80493,82108,43801,4293,118276,78521
C01029=-80495,81630,46278,4216,116511,78452
C01030=-80492,84058,47940,4226,116735,78462
C01031=-83493,53381,-2692,9637,111099,78940
C01032=-91945,-14209,-43630,9790,83010,75128
C01033=-10907,-117335,-90652,-18762,63715,-59495
C01034=-15972,-110889,-128286,-10965,59905,-43045
BC00000=48829,688840,1075175
BC00001=366911,902233,1075175
BC00002=366911,902233,1075175
BC00003=366911,902233,1075175
BC00004=366911,902233,1075175
BC00005=366911,902233,1075175
BC00006=366911,902233,1075175
BC00007=366911,902233,1075175
BC00008=366911,902233,1075175
BC00009=333056,895412,1075175
BC00010=333056,895412,1075175
BC00011=333056,895412,1075175
BC00012=333056,895412,1075175
BC00013=333056,895412,1075175
BC00014=333056,895412,1075175
BC00015=333056,895412,1075175
BC00016=333056,895412,1075175
BC00017=358091,902222,1075175
BC00018=358091,902222,1075175
BC00019=358091,902222,1075175
BC00020=358091,902222,1075175
BC00021=358091,902222,1075175
BC00022=358091,902222,1075175
BC00023=358091,902222,1075175
BC00024=358091,902222,1075175
BC00025=398174,894103,1075175
BC00026=398174,894103,1075175
BC00027=398174,894103,1075175
BC00028=398174,894103,1075175
BC00029=398174,894103,1075175
BC00030=398174,894103,1075175
BC00031=398174,894103,1075175
BC00032=398174,894103,1075175
BC00033=264903,781270,1075175
BC00034=264903,781270,1075175
BC00035=264904,781269,1075172
BC00036=264904,781269,1075171
BC00037=264904,781269,1075171
BC00038=264904,781269,1075168
BC00039=264904,781269,1075168
BC00040=264904,781269,1075168
BC00041=264904,781269,1075168
BC00042=264904,781269,1075168
BC00043=264904,781269,1075164
BC00044=264903,781270,1075175
BC00045=301264,775814,1075175
BC00046=301264,775814,1075175
BC00047=301264,775814,1075175
BC00048=301264,775814,1075175
BC00049=301264,775814,1075175
BC00050=301264,775814,1075175
BC00051=301264,775814,1075175
BC00052=301264,775814,1075175
BC00053=301264,775814,1075175
BC00054=301264,775814,1075175
BC00055=274235,786209,1075175
BC00056=238672,799885,1075175
BC00057=238672,799885,1075175
BC00058=238672,799885,1075175
BC00059=238672,799885,1075175
BC00060=238672,799885,1075175
BC00061=238672,799885,1075175
BC00062=238672,799885,1075175
BC00063=238672,799885,1075175
BC00064=238672,799884,1075171
BC00065=238672,799884,1075171
BC00066=238672,799885,1075175
BC00067=238672,799885,1075175
BC00068=238672,799885,1075175
BC00069=238672,799885,1075175
BC00070=318263,750454,1075175
BC00071=318263,750454,1075175
BC00072=318263,750454,1075175
BC00073=318263,750454,1075175
BC00074=318263,750454,1075175
BC00075=318263,750454,1075175
BC00076=318263,750454,1075175
BC00077=318263,750454,1075175
BC00078=318263,750454,1075175
BC00079=318263,750454,1075175
BC00080=318263,750454,1075175
BC00081=318263,750454,1075175
BC00082=318263,750454,1075175
BC00083=318263,750454,1075175
BC00084=318263,750454,1075175
BC00085=318263,750454,1075175
BC00086=318263,750454,1075175
BC00087=318263,750454,1075175
BC00088=318263,750454,1075175
BC00089=318263,750454,1075175
BC00090=318263,750454,1075175
BC00091=318263,750454,1075175
BC00092=318263,750454,1075175
BC00093=318263,750454,1075175
BC00094=318263,750454,1075175
BC00095=377114,750454,1075175
BC00096=397814,750454,1075175
BC00097=397814,750454,1075175
BC00098=397814,750454,1075175
BC00099=397814,750454,1075175
BC00100=397814,750454,1075175
BC00101=397814,750454,1075175
BC00102=397814,750454,1075175
BC00103=397814,750454,1075175
BC00104=397814,750454,1075175
BC00105=397814,750454,1075175
BC00106=397814,750454,1075175
BC00107=397814,750454,1075175
BC00108=397814,750454,1075175
BC00109=397814,750454,1075175
BC00110=397814,750454,1075175
BC00111=397814,750454,1075175
BC00112=397814,750454,1075175
BC00113=397814,750454,1075175
BC00114=397814,750454,1075175
BC00115=397814,750454,1075175
BC00116=383090,762961,1075175
BC00117=372387,772052,1075175
BC00118=296274,836703,1075175
BC00119=296274,836703,1075175
BC00120=296274,836703,1075175
BC00121=296274,836703,1075175
BC00122=296274,836703,1075175
BC00123=296274,836703,1075175
BC00124=296274,836703,1075175
BC00125=296274,836703,1075175
BC00126=296274,836703,1075175
BC00127=296274,836703,1075175
BC00128=296274,836703,1075175
BC00129=296274,836703,1075175
BC00130=296274,836703,1075175
BC00131=312215,899988,1075175
BC00132=312215,944285,1075175
BC00133=312215,944285,1075175
BC00134=312215,944285,1075175
BC00135=312215,944285,1075175
BC00136=312215,944285,1075175
BC00137=312215,944285,1075175
BC00138=312215,944285,1075175
BC00139=312215,944285,1075175
BC00140=312215,944285,1075175
BC00141=312215,944285,1075175
BC00142=312215,944285,1075175
BC00143=259299,938961,1075175
BC00144=259299,938961,1075175
BC00145=259299,938961,1075175
BC00146=259299,938961,1075175
BC00147=259299,938961,1075175
BC00148=259299,938961,1075175
BC00149=259299,938961,1075175
BC00150=259299,938961,1075175
BC00151=259299,938961,1075175
BC00152=259299,938961,1075175
BC00153=259299,938961,1075175
BC00154=259299,938961,1075175
BC00155=211531,951911,1075175
BC00156=211531,951911,1075175
BC00157=211531,951911,1075175
BC00158=211531,951911,1075175
BC00159=211531,951911,1075175
BC00160=211531,951911,1075175
BC00161=211531,951911,1075175
BC00162=211531,951911,1075175
BC00163=211531,951911,1075175
BC00164=211531,951911,1075175
BC00165=211531,951911,1075175
BC00166=182503,951872,1075175
BC00167=184369,953383,1075175
BC00168=184369,953399,1075175
BC00169=184333,953526,1075175
BC00170=184897,956550,1075175
BC00171=184333,953526,1075175
BC00172=184751,953664,1075175
BC00173=187887,953121,1075175
BC00174=184751,953664,1075175
BC00175=178222,948378,1075175
BC00176=171711,951911,1075175
BC00177=171711,959591,1075175
BC00178=171711,959591,1075175
BC00179=171711,959591,1075175
BC00180=171711,959591,1075175
BC00181=171711,959591,1075175
BC00182=171711,959591,1075175
BC00183=171711,959591,1075175
BC00184=171711,959591,1075175
BC00185=171711,959591,1075175
BC00186=182815,952263,1075175
BC00187=183711,957103,1075175
BC00188=184069,959047,1075174
BC00189=184070,959056,1075175
BC00190=184189,959079,1075175
BC00191=184752,962103,1075175
BC00192=184189,959079,1075175
BC00193=182935,952303,1075175
BC00194=148303,998123,1075175
BC00195=123088,1061215,1075175
BC00196=126332,1055781,1075175
BC00197=127630,1053613,1075175
BC00198=127630,1053623,1075175
BC00199=127630,1053607,1075175
BC00200=153753,1064749,1075175
BC00201=152152,1062093,1075175
BC00202=153753,1064749,1075175
BC00203=104366,1038154,1075175
BC00204=107120,1036610,1075175
BC00205=104366,1038154,1075175
BC00206=97490,1044180,1075175
BC00207=121157,1044973,1075175
BC00208=140343,1045718,1075175
BC00209=158643,1046375,1075175
BC00210=155464,1041036,1075175
BC00211=155106,1040455,1075175
BC00212=155106,1040463,1075175
BC00213=155288,1040367,1075175
BC00214=153687,1037711,1075175
BC00215=155288,1040367,1075175
BC00216=158891,1046297,1075175
BC00217=211337,993614,1075175
BC00218=274623,983932,1075175
BC00219=371761,1043051,1075175
BC00220=331941,1063020,1075175
BC00221=331941,1063020,1075175
BC00222=331941,1063020,1075175
BC00223=331941,1063020,1075175
BC00224=331941,1063020,1075175
BC00225=331941,1063020,1075175
BC00226=331941,1063020,1075175
BC00227=331941,1063020,1075175
BC00228=331941,1063020,1075175
BC00229=331941,1063020,1075175
BC00230=331941,1063020,1075175
BC00231=331941,1063020,1075175
BC00232=331941,1063020,1075175
BC00233=371761,1043051,1075175
BC00234=371761,1043051,1075175
BC00235=371761,1043051,1075175
BC00236=371761,1043051,1075175
BC00237=371761,1043051,1075175
BC00238=371761,1043051,1075175
BC00239=371761,1043051,1075175
BC00240=371761,1043051,1075175
BC00241=371761,1043051,1075175
BC00242=371761,1043051,1075175
BC00243=371761,1043051,1075175
BC00244=371761,1043051,1075175
BC00245=371761,1043051,1075175
BC00246=371761,1043051,1075175
BC00247=371761,1043051,1075175
BC00248=314185,938855,1075175
BC00249=247671,970611,1075175
BC00250=247671,970611,1075175
BC00251=247671,970611,1075175
BC00252=247671,970611,1075175
BC00253=247671,970611,1075175
BC00254=247671,970611,1075175
BC00255=247671,970611,1075175
BC00256=247671,970611,1075175
BC00257=247671,970611,1075175
BC00258=247671,970611,1075175
BC00259=247671,970611,1075175
BC00260=247671,970611,1075175
BC00261=303037,872055,1075175
BC00262=380992,820655,1075175
BC00263=380992,820655,1075175
BC00264=380992,820655,1075175
BC00265=380992,820655,1075175
BC00266=380992,820655,1075175
BC00267=380992,820655,1075175
BC00268=380992,820655,1075175
BC00269=380992,820655,1075175
BC00270=380992,820655,1075175
BC00271=380992,820655,1075175
BC00272=380992,820655,1075175
BC00273=380992,820655,1075175
BC00274=275256,812324,1075175
BC00275=125716,897903,1075175
BC00276=125716,897903,1075175
BC00277=125716,897903,1075175
BC00278=125716,897903,1075175
BC00279=125716,897903,1075175
BC00280=125716,897903,1075174
BC00281=125716,897903,1075171
BC00282=125716,897903,1075175
BC00283=125716,897903,1075175
BC00284=125716,897903,1075175
BC00285=125716,897903,1075175
BC00286=125716,897903,1075175
BC00287=125716,897903,1075175
BC00288=325019,822543,1075229
BC00289=325019,822543,1075229
BC00290=325019,822543,1075229
BC00291=325019,822543,1075229
BC00292=325019,822543,1075229
BC00293=325019,822543,1075229
BC00294=325019,822543,1075229
BC00295=325019,822543,1075229
BC00296=325019,822543,1075229
BC00297=325019,822543,1075229
BC00298=325019,822543,1075229
BC00299=325019,822543,1075229
BC00300=240667,871930,1075210
BC00301=81335,965219,1075175
BC00302=81335,965219,1075175
BC00303=81335,965219,1075175
BC00304=81335,965219,1075175
BC00305=81335,965219,1075175
BC00306=81335,965219,1075175
BC00307=81335,965219,1075175
BC00308=81335,965219,1075175
BC00309=39891,972466,1075175
BC00310=39891,972466,1075175
BC00311=39891,972466,1075175
BC00312=39891,972466,1075175
BC00313=39891,972466,1075175
BC00314=39891,972466,1075175
BC00315=39891,972466,1075175
BC00316=39891,972466,1075175
BC00317=126064,942124,1075175
BC00318=145718,951183,1075175
BC00319=145718,951183,1075175
BC00320=145718,951183,1075175
BC00321=145718,951183,1075175
BC00322=145718,951183,1075175
BC00323=145718,951183,1075175
BC00324=145718,951183,1075175
BC00325=145718,951183,1075175
BC00326=145718,951183,1075175
BC00327=145718,951183,1075175
BC00328=145718,951183,1075175
BC00329=145718,951183,1075175
BC00330=127193,914007,1075175
BC00331=75497,867475,1075175
BC00332=75497,867475,1075175
BC00333=75497,867475,1075175
BC00334=75497,867475,1075175
BC00335=75497,867475,1075175
BC00336=75497,867475,1075175
BC00337=75497,867475,1075175
BC00338=75497,867475,1075175
BC00339=75497,867475,1075175
BC00340=75497,867475,1075175
BC00341=75497,867475,1075175
BC00342=75497,867475,1075175
BC00343=75497,867475,1075175
BC00344=75497,867475,1075175
BC00345=75497,867475,1075175
BC00346=75497,867475,1075175
BC00347=75497,867475,1075175
BC00348=58830,852413,1075175
BC00349=43274,838354,1075175
BC00350=43274,838354,1075175
BC00351=43274,838354,1075175
BC00352=43274,838354,1075175
BC00353=43274,838354,1075175
BC00354=43274,838354,1075175
BC00355=43274,838354,1075175
BC00356=43274,838354,1075175
BC00357=43274,838354,1075175
BC00358=191439,896290,1075175
BC00359=209593,874493,1075175
BC00360=209593,874493,1075175
BC00361=209593,874493,1075175
BC00362=209593,874493,1075171
BC00363=209593,874493,1075175
BC00364=209593,874493,1075175
BC00365=209216,850926,1075175
BC00366=226866,854473,1075175
BC00367=228835,855864,1075175
BC00368=228835,855864,1075175
BC00369=228834,855864,1075173
BC00370=228834,855864,1075173
BC00371=228835,855864,1075175
BC00372=228835,855864,1075175
BC00373=228835,855864,1075175
BC00374=228835,855864,1075175
BC00375=228835,855864,1075175
BC00376=212683,986357,1075175
BC00377=212683,1004517,1075175
BC00378=212247,999872,1075175
BC00379=212146,998778,1075171
BC00380=214955,996593,1075174
BC00381=222186,994128,1075175
BC00382=222622,998773,1075175
BC00383=293477,973063,1075175
BC00384=293477,973063,1075175
BC00385=293477,973063,1075175
BC00386=293477,973063,1075175
BC00387=293477,973063,1075175
BC00388=293477,973063,1075175
BC00389=293477,973063,1075175
BC00390=293477,973063,1075175
BC00391=248777,974412,1075175
BC00392=147624,1017934,1075175
BC00393=124950,1033375,1075175
BC00394=124950,1033375,1075175
BC00395=124950,1033375,1075175
BC00396=124950,1033375,1075175
BC00397=124950,1033375,1075175
BC00398=124950,1033375,1075175
BC00399=106678,1046165,1075175
BC00400=106678,1046165,1075175
BC00401=106678,1046165,1075175
BC00402=106678,1046165,1075175
BC00403=106678,1046165,1075175
BC00404=106678,1046165,1075175
BC00405=172863,1024486,1075175
BC00406=172427,1019841,1075175
BC00407=172326,1018747,1075171
BC00408=175135,1016562,1075174
BC00409=182366,1014097,1075175
BC00410=182802,1018742,1075175
BC00411=253657,993032,1075175
BC00412=253657,993032,1075175
BC00413=253657,993032,1075175
BC00414=253657,993032,1075175
BC00415=253657,993032,1075175
BC00416=253657,993032,1075175
BC00417=253657,993032,1075175
BC00418=253657,993032,1075175
BC00419=208957,994381,1075175
BC00420=107804,1037903,1075175
BC00421=85130,1053344,1075175
BC00422=85130,1053344,1075175
BC00423=85130,1053344,1075175
BC00424=85130,1053344,1075175
BC00425=85130,1053344,1075175
BC00426=85130,1053344,1075175
BC00427=66858,1066134,1075175
BC00428=66858,1066134,1075175
BC00429=66858,1066134,1075175
BC00430=66858,1066134,1075175
BC00431=66858,1066134,1075175
BC00432=66858,1066134,1075175
BC00433=106678,1034404,1075175
BC00434=288363,951317,1075175
BC00435=319880,932288,1075175
BC00436=316203,930177,1075175
BC00437=314732,929332,1075175
BC00438=314732,929332,1075175
BC00439=294141,940882,1075175
BC00440=285351,949486,1075175
BC00441=280844,953897,1075175
BC00442=254356,968931,1075172
BC00443=253996,970793,1075175
BC00444=256777,973747,1075175
BC00445=224914,994659,1075175
BC00446=193407,1014756,1075175
BC00447=196552,1009267,1075175
BC00448=197065,1008372,1075175
BC00449=197397,1007797,1075175
BC00450=196552,1009278,1075175
BC00451=193407,1014766,1075175
BC00452=170876,1031134,1075175
BC00453=153007,1044116,1075175
BC00454=153007,1044116,1075175
BC00455=155599,1038213,1075175
BC00456=156636,1035851,1075175
BC00457=230598,1025728,1075175
BC00458=222023,1030515,1075175
BC00459=222023,1030515,1075175
BC00460=118655,1062836,1075175
BC00461=118655,1062836,1075175
BC00462=118655,1062836,1075175
BC00463=176896,1055708,1075175
BC00464=225377,1010635,1075175
BC00465=228184,1010601,1075175
BC00466=235201,1010515,1075175
BC00467=242597,980334,1075175
BC00468=282680,816770,1075175
BC00469=287393,774165,1075175
BC00470=293866,776192,1075175
BC00471=296455,777002,1075175
BC00472=296337,777088,1075175
BC00473=296308,777110,1075175
BC00474=296189,777197,1075175
BC00475=293600,776386,1075175
BC00476=287127,774359,1075175
BC00477=265173,805126,1075175
BC00478=271841,806848,1075175
BC00479=274508,807537,1075175
BC00480=274508,807537,1075175
BC00481=271842,806893,1075175
BC00482=265174,805171,1075175
BC00483=347775,809657,1075175
BC00484=348436,809459,1075175
BC00485=348700,809380,1075175
BC00486=352833,807067,1075175
BC00487=364813,800347,1075175
BC00488=368942,798027,1075175
BC00489=368677,798106,1075175
BC00490=368016,798304,1075175
BC00491=368016,798304,1075175
BC00492=391344,687000,1075175
BC00493=391344,687000,1075175
BC00494=391344,687000,1075175
BC00495=391344,687000,1075175
BC00496=391344,687000,1075175
BC00497=391344,687000,1075175
BC00498=391344,687000,1075175
BC00499=391344,687000,1075175
BC00500=391344,687000,1075175
BC00501=391344,687000,1075175
BC00502=391344,687000,1075175
BC00503=391344,687000,1075175
BC00504=358873,687000,1075175
BC00505=250171,896024,1075175
BC00506=255370,893912,1075175
BC00507=257449,893067,1075175
BC00508=259851,897051,1075175
BC00509=270502,914711,1075175
BC00510=268422,915555,1075175
BC00511=263223,917668,1075175
BC00512=251695,824506,1075175
BC00513=253916,829548,1075175
BC00514=254804,831565,1075175
BC00515=231448,844598,1075175
BC00516=231448,844598,1075175
BC00517=189878,862044,1075175
BC00518=188570,860127,1075175
BC00519=185301,855336,1075175
BC00520=261332,833542,1075175
BC00521=297112,823286,1075175
BC00522=293523,829343,1075175
BC00523=292087,831765,1075175
BC00524=292088,831788,1075175
BC00525=293523,829365,1075175
BC00526=297112,823308,1075175
BC00527=297112,823286,1075175
BC00528=112345,954746,1075175
BC00529=112345,954746,1075175
BC00530=111546,959512,1075175
BC00531=111226,961418,1075175
BC00532=63698,969650,1075175
BC00533=64018,967744,1075175
BC00534=64817,962978,1075175
BC00535=55529,859309,1075175
BC00536=51595,858048,1075175
BC00537=50021,857544,1075175
BC00538=45895,833192,1075175
BC00539=46071,849801,1075175
BC00540=43912,844296,1075175
BC00541=45475,843733,1075175
BC00542=45475,843733,1075175
BC00543=45475,843733,1075175
BC00544=45475,843733,1075175
BC00545=45475,843733,1075175
BC00546=49382,842326,1075175
BC00547=32191,855540,1075175
BC00548=35199,856902,1075175
BC00549=36402,857447,1075175
BC00550=24170,872455,1075175
BC00551=24116,855865,1075175
BC00552=17601,856883,1075175
BC00553=10106,858388,1075175
BC00554=7107,859694,1075175
BC00555=124165,958731,1075175
BC00556=124477,964204,1075175
BC00557=124602,966393,1075175
BC00558=119899,967208,1075175
BC00559=114659,968116,1075175
BC00560=114534,965927,1075175
BC00561=114222,960453,1075175
BC00562=169497,963360,1075175
BC00563=218455,965934,1075175
BC00564=214431,967961,1075175
BC00565=212822,968772,1075175
BC00566=212822,968772,1075175
BC00567=212822,968772,1075175
BC00568=212822,968772,1075175
BC00569=218344,963319,1075175
BC00570=222368,961291,1075175
BC00571=147324,958268,1075175
BC00572=86350,984014,1075175
BC00573=90717,985390,1075175
BC00574=92241,985755,1075175
BC00575=87949,982178,1075175
BC00576=87949,982178,1075175
BC00577=87949,982178,1075175
BC00578=86202,981627,1075175
BC00579=81835,980250,1075175
BC00580=83182,969192,1075175
BC00581=84657,971884,1075175
BC00582=84782,974073,1075175
BC00583=80079,974888,1075175
BC00584=74839,975796,1075175
BC00585=74714,973607,1075175
BC00586=74402,968133,1075175
BC00587=129677,971040,1075175
BC00588=178635,973614,1075175
BC00589=174611,975641,1075175
BC00590=173002,976452,1075175
BC00591=173002,976452,1075175
BC00592=173002,976452,1075175
BC00593=173002,976452,1075175
BC00594=178524,970999,1075175
BC00595=182548,968971,1075175
BC00596=107504,965948,1075175
BC00597=46530,991694,1075175
BC00598=50897,993070,1075175
BC00599=52421,993435,1075175
BC00600=48129,989858,1075175
BC00601=48129,989858,1075175
BC00602=48129,989858,1075175
BC00603=46382,989307,1075175
BC00604=42015,987930,1075175
BC00605=86350,984014,1075175
BC00606=118186,882849,1075175
BC00607=118313,879045,1075175
BC00608=118363,877523,1075175
BC00609=127351,877496,1075175
BC00610=127300,879018,1075175
BC00611=127173,882822,1075175
BC00612=149531,895732,1075175
BC00613=148249,891267,1075175
BC00614=148034,889482,1075175
BC00615=151775,889498,1075175
BC00616=152288,891284,1075175
BC00617=153569,895750,1075175
BC00618=119302,902119,1075175
BC00619=119440,897649,1075175
BC00620=119495,895861,1075175
BC00621=115974,895890,1075175
BC00622=115919,897678,1075175
BC00623=115781,902148,1075175
BC00624=206850,915693,1075175
BC00625=246637,921611,1075175
BC00626=251241,924622,1075175
BC00627=253082,925827,1075175
BC00628=305626,902567,1075175
BC00629=289523,905356,1075175
BC00630=289523,905356,1075175
BC00631=265997,901694,1075172
BC00632=265782,900020,1075175
BC00633=265246,895833,1075175
BC00634=152805,918674,1075175
BC00635=155644,922700,1075175
BC00636=156780,924310,1075175
BC00637=187141,913105,1075175
BC00638=179441,914454,1075175
BC00639=179441,914454,1075175
BC00640=179441,914454,1075175
BC00641=120688,931609,1075175
BC00642=120688,931609,1036122
BC00643=120688,931609,1036122
BC00644=135499,922155,1075175
BC00645=196755,924293,1075175
BC00646=204603,922909,1075175
BC00647=210067,918954,1075175
BC00648=285493,836258,1075175
BC00649=322674,778579,1075175
BC00650=322674,778579,1075175
BC00651=322674,778579,1075175
BC00652=322674,778579,1075175
BC00653=322674,778579,1075175
BC00654=322674,778579,1075175
BC00655=322674,778579,1075175
BC00656=322674,778579,1075175
BC00657=272555,769164,1075175
BC00658=266479,768023,1075175
BC00659=266479,768023,1075175
BC00660=267479,770239,1071365
BC00661=266799,769335,1075175
BC00662=266479,768023,1075175
BC00663=266479,768023,1075175
BC00664=266479,768023,1075175
BC00665=266479,768023,1075175
BC00666=235984,786404,1075175
BC00667=235984,786404,1075175
BC00668=235984,786404,1075175
BC00669=235984,786404,1075175
BC00670=235984,786404,1075175
BC00671=235984,786404,1075175
BC00672=235984,786404,1075175
BC00673=235984,786404,1075175
BC00674=237203,787368,1075175
BC00675=295022,827394,1075175
BC00676=205701,931185,1075175
BC00677=204812,932218,1075175
BC00678=205671,937629,1075175
BC00679=206015,939793,1075175
BC00680=202546,941762,1075175
BC00681=218293,952795,1075175
BC00682=218466,950486,1075175
BC00683=218898,944716,1075175
BC00684=188226,925402,1075175
BC00685=189298,932104,1075175
BC00686=189728,934784,1075175
BC00687=185375,937227,1075175
BC00688=184946,934546,1075175
BC00689=183874,927845,1075175
BC00690=163256,940528,1075175
BC00691=166760,944877,1075175
BC00692=168161,946617,1075175
BC00693=172960,943924,1075175
BC00694=171559,942185,1075175
BC00695=168055,937836,1075175
BC00696=205604,952176,1075175
BC00697=237375,964309,1075175
BC00698=234858,970014,1075175
BC00699=233851,972296,1075175
BC00700=237408,970622,1075175
BC00701=238426,968449,1075175
BC00702=241139,962660,1075175
BC00703=186195,958850,1075175
BC00704=137530,955476,1075175
BC00705=142340,959691,1075175
BC00706=135217,966057,1075175
BC00707=135217,966057,1075175
BC00708=134381,966543,1075175
BC00709=132263,964948,1075175
BC00710=126968,960962,1075175
BC00711=137530,955476,1075175
BC00712=284870,850327,1075175
BC00713=323104,941595,1075175
BC00714=324436,944989,1075175
BC00715=324969,946346,1075175
BC00716=379859,936839,1075175
BC00717=379326,935482,1075175
BC00718=377994,932088,1075175
BC00719=387025,925803,1075175
BC00720=391871,922431,1075175
BC00721=387133,926188,1075175
BC00722=385238,927691,1075175
BC00723=381091,925537,1075175
BC00724=365308,912570,1075175
BC00725=363166,908743,1075175
BC00726=364796,906869,1075175
BC00727=368870,902183,1075175
BC00728=358157,902408,1075175
BC00729=354876,908652,1075175
BC00730=353564,911150,1075175
BC00731=349138,907302,1075175
BC00732=357572,916934,1075175
BC00733=359178,914754,1075175
BC00734=363193,909304,1075175
BC00735=322758,853588,1075175
BC00736=135439,955204,1075175
BC00737=139952,957848,1075175
BC00738=141757,958906,1075175
BC00739=133040,997822,1075175
BC00740=133065,977483,1075175
BC00741=144047,1040883,1075175
BC00742=142698,1043050,1075175
BC00743=139327,1048468,1075175
BC00744=139327,1048468,1075175
BC00745=95619,955204,1075175
BC00746=100132,965528,1075175
BC00747=101937,966586,1075175
BC00748=93220,1005502,1075175
BC00749=93220,1005502,1075175
BC00750=93221,1030527,1075216
BC00751=93221,1030527,1075216
BC00752=99566,1045795,1075190
BC00753=142698,1043050,1075175
BC00754=206177,1018673,1075175
BC00755=252443,1048931,1075175
BC00756=258757,1029159,1075175
BC00757=290253,930536,1075175
BC00758=290253,930536,1075175
BC00759=290253,930536,1075175
BC00760=297151,966120,1075172
BC00761=297151,997903,1075172
BC00762=297151,997903,1075172
BC00763=297194,1021413,1075172
BC00764=297194,1021413,1075172
BC00765=21214,672831,1075175
BC00766=21214,672831,429902
BC00767=66815,724118,419761
BC00768=110240,772957,337669
BC00769=124996,789553,122283
BC00770=124996,789553,122283
BC00771=124996,789553,122283
BC00772=124996,789553,122283
BC00773=124996,789553,122283
BC00774=124996,789553,122283
BC00775=124996,789553,122283
BC00776=124996,789553,122283
BC00777=124996,789553,122283
BC00778=124996,789553,122283
BC00779=136729,789553,283981
BC00780=136729,789553,283981
BC00781=136729,789553,283981
BC00782=136729,789553,283981
BC00783=136729,789553,283981
BC00784=136729,789553,283981
BC00785=136729,789553,283981
BC00786=136729,789553,283981
BC00787=136729,789553,283981
BC00788=136729,789553,283981
BC00789=163194,789553,386705
BC00790=163194,789553,386705
BC00791=163194,789553,386705
BC00792=163194,789553,386705
BC00793=163194,789553,386705
BC00794=163194,789553,386705
BC00795=163194,789553,386705
BC00796=163194,789553,386705
BC00797=163194,789553,386705
BC00798=163194,789553,386705
BC00799=110240,772957,337669
BC00800=66815,724118,419761
BC00801=66815,670858,419761
BC00802=252765,670858,277331
BC00803=322808,760288,131711
BC00804=322808,760288,131711
BC00805=322808,760288,131711
BC00806=322808,760288,131711
BC00807=322808,760288,131711
BC00808=322808,760288,131711
BC00809=322808,760288,131711
BC00810=322808,760288,131711
BC00811=322808,760288,131711
BC00812=335534,789553,204922
BC00813=335534,789553,204922
BC00814=335534,789553,204922
BC00815=335534,789553,204922
BC00816=335534,789553,204922
BC00817=335534,789553,204922
BC00818=335534,789553,204922
BC00819=335534,789553,204922
BC00820=335534,789553,204922
BC00821=344006,752651,139062
BC00822=344006,752651,139062
BC00823=344006,752651,139062
BC00824=344006,752651,139062
BC00825=344006,752651,139062
BC00826=344006,752651,139062
BC00827=344006,752651,139062
BC00828=344006,752651,139062
BC00829=344006,752651,139062
BC00830=300933,750795,218908
BC00831=283893,750061,250495
BC00832=276320,749735,264534
BC00833=276320,749735,264534
BC00834=276320,749735,264534
BC00835=276320,749735,264534
BC00836=276320,749735,264534
BC00837=276320,749735,264534
BC00838=276320,749735,264534
BC00839=276320,749735,264534
BC00840=276320,749735,264534
BC00841=248857,763770,138691
BC00842=248857,763770,138691
BC00843=248857,763770,138691
BC00844=248857,763770,138691
BC00845=248857,763770,138691
BC00846=248857,763770,138691
BC00847=248857,763770,138691
BC00848=248857,763770,138691
BC00849=248857,763770,138691
BC00850=287864,789553,132710
BC00851=287864,789553,132710
BC00852=287864,789553,132710
BC00853=287864,789553,132710
BC00854=287864,789553,132710
BC00855=287864,789553,132710
BC00856=287864,789553,132710
BC00857=287864,789553,132710
BC00858=287864,789553,132710
BC00859=287864,789553,132710
BC00860=287864,789553,132710
BC00861=287864,789553,132710
BC00862=279829,789553,53
BC00863=279829,789553,53
BC00864=279829,789553,53
BC00865=279829,789553,53
BC00866=279829,789553,53
BC00867=279829,789553,53
BC00868=279829,789553,53
BC00869=279829,789553,53
BC00870=279829,789553,53
BC00871=279829,789553,53
BC00872=279829,789553,53
BC00873=279829,789553,53
BC00874=279829,789553,53
BC00875=312324,789553,158805
BC00876=312324,789553,158805
BC00877=312324,789553,158804
BC00878=312324,789553,158805
BC00879=312324,789553,158805
BC00880=312324,789553,158805
BC00881=303082,768394,105099
BC00882=303082,768394,105099
BC00883=303082,768394,105099
BC00884=303082,768394,105099
BC00885=303082,768394,105099
BC00886=303082,768394,105099
BC00887=287868,781442,183325
BC00888=278410,789553,231953
BC00889=278410,789553,231953
BC00890=278410,789553,231953
BC00891=278410,789553,231953
BC00892=278410,789553,231953
BC00893=278410,789553,231953
BC00894=283893,750061,250495
BC00895=300933,750795,218908
BC00896=376723,772526,120737
BC00897=376723,772526,120737
BC00898=376723,772526,120737
BC00899=376723,772526,120737
BC00900=376723,772526,120737
BC00901=376723,772526,120737
BC00902=385013,737075,95404
BC00903=385013,737075,95404
BC00904=385013,737075,95404
BC00905=385013,737075,95404
BC00906=385013,737075,95404
BC00907=385013,737075,95404
BC00908=365962,760163,122379
BC00909=365962,760163,122379
BC00910=365962,760163,122379
BC00911=365962,760163,122379
BC00912=365962,760163,122379
BC00913=365962,760163,122379
BC00914=365962,760163,122379
BC00915=252765,670858,277331
BC00916=66815,670858,419761
BC00917=66815,724118,419761
BC00918=110240,772957,337669
BC00919=118803,789553,240458
BC00920=118803,789553,240458
BC00921=118803,789553,240458
BC00922=118803,789553,240458
BC00923=118803,789553,240458
BC00924=118803,789553,240458
BC00925=130259,789553,198376
BC00926=110709,789553,198376
BC00927=113251,789553,198376
BC00928=113251,789553,198376
BC00929=113251,789553,198376
BC00930=113251,789553,198376
BC00931=113251,789553,198376
BC00932=113251,789553,198376
BC00933=113251,789553,198376
BC00934=113251,789553,198376
BC00935=113251,789553,198376
BC00936=113251,789553,198376
BC00937=113251,789553,198376
BC00938=113251,789553,198376
BC00939=113251,789553,198376
BC00940=113251,789553,228042
BC00941=113251,789553,280292
BC00942=113251,789553,280290
BC00943=113251,789553,280290
BC00944=113251,789553,280290
BC00945=113251,789553,280290
BC00946=113251,789553,280290
BC00947=113251,789553,280290
BC00948=113251,789553,280290
BC00949=110240,772957,337669
BC00950=66815,724118,419761
BC00951=66815,670858,419761
BC00952=252765,670858,277331
BC00953=298333,782774,240815
BC00954=298333,782774,240815
BC00955=298333,782774,240815
BC00956=298333,782774,240815
BC00957=298333,782774,240815
BC00958=298333,782774,240815
BC00959=277596,773081,190929
BC00960=277596,773081,190929
BC00961=277596,773081,190929
BC00962=277596,773081,190929
BC00963=277596,773081,190929
BC00964=277596,773081,190929
BC00965=252765,670858,277331
BC00966=66815,670858,419761
BC00967=66815,724118,419761
BC00968=110240,772957,337669
BC00969=116545,789553,319269
BC00970=116545,789553,319269
BC00971=116545,789553,319269
BC00972=116545,789553,319269
BC00973=116545,789553,319269
BC00974=116545,789553,319269
BC00975=104258,789553,379308
BC00976=104258,789553,379308
BC00977=104258,789553,379308
BC00978=104258,789553,379308
BC00979=104258,789553,379308
BC00980=104258,789553,379308
BC00981=110240,772957,337669
BC00982=66815,724118,419761
BC00983=66815,670858,419761
BC00984=252765,670858,277331
BC00985=286674,787255,240962
BC00986=286675,787255,240962
BC00987=286675,787255,240962
BC00988=286675,787255,240962
BC00989=286674,787255,240962
BC00990=286674,787255,240962
BC00991=267109,758037,158941
BC00992=267109,758037,158941
BC00993=267109,758037,158941
BC00994=267109,758037,158941
BC00995=267109,758037,158941
BC00996=267109,758037,158941
BC00997=283893,750061,250495
BC00998=360336,760725,110934
BC00999=360336,760725,110934
BC01000=360336,760725,110934
BC01001=360336,760725,110934
BC01002=360336,760725,110934
BC01003=360336,760725,110934
BC01004=371149,789553,191296
BC01005=371149,789553,191296
BC01006=371149,789553,191296
BC01007=371149,789553,191296
BC01008=371149,789553,191296
BC01009=371149,789553,191296
BC01010=283893,750061,250495
BC01011=292970,789553,136523
BC01012=292970,789553,136523
BC01013=292970,789553,136523
BC01014=292970,789553,136523
BC01015=292970,789553,136523
BC01016=292970,789552,136519
BC01017=292970,789553,136523
BC01018=292970,789553,136523
BC01019=256495,759418,21571
BC01020=256495,759418,21571
BC01021=256495,759418,21571
BC01022=256495,759418,21571
BC01023=256495,759418,21571
BC01024=256495,759418,21571
BC01025=256075,748610,41729
BC01026=255916,738170,60084
BC01027=255916,738170,60084
BC01028=255916,738170,60084
BC01029=255916,738170,60084
BC01030=255916,738170,60084
BC01031=255916,738170,60084
BC01032=262339,748900,193466
BC01033=165820,667836,534036
BC01034=21214,672831,1075175
EC00000=798156,1112951
EC00001=798156,1112951
EC00002=798156,1112951
EC00003=798156,1112951
EC00004=798156,1112951
EC00005=798156,1112951
EC00006=798156,1112951
EC00007=798156,1112951
EC00008=798156,1112951
EC00009=798156,1112951
EC00010=798156,1112951
EC00011=798156,1112951
EC00012=798156,1112951
EC00013=798156,1112951
EC00014=798156,1112951
EC00015=798156,1112951
EC00016=798156,1112951
EC00017=798156,1112951
EC00018=798156,1112951
EC00019=798156,1112951
EC00020=798156,1112951
EC00021=798156,1112951
EC00022=798156,1112951
EC00023=798156,1112951
EC00024=798156,1112951
EC00025=798156,1112951
EC00026=798156,1112951
EC00027=798156,1112951
EC00028=798156,1112951
EC00029=798156,1112951
EC00030=798156,1112951
EC00031=798156,1112951
EC00032=798156,1112951
EC00033=798156,1112951
EC00034=798156,1112951
EC00035=798155,1112950
EC00036=798155,1112950
EC00037=798155,1112950
EC00038=798154,1112949
EC00039=798154,1112949
EC00040=798154,1112949
EC00041=798154,1112949
EC00042=798154,1112949
EC00043=798153,1112949
EC00044=798156,1112951
EC00045=798156,1112951
EC00046=798156,1112951
EC00047=798156,1112951
EC00048=798156,1112951
EC00049=798156,1112951
EC00050=798156,1112951
EC00051=798156,1112951
EC00052=798156,1112951
EC00053=798156,1112951
EC00054=798156,1112951
EC00055=798156,1112951
EC00056=798156,1112951
EC00057=798156,1112951
EC00058=798156,1112951
EC00059=798156,1112951
EC00060=798156,1112951
EC00061=798156,1112951
EC00062=798156,1112951
EC00063=798156,1112951
EC00064=798155,1112950
EC00065=798155,1112950
EC00066=798156,1112951
EC00067=798156,1112951
EC00068=798156,1112951
EC00069=798156,1112951
EC00070=798156,1112951
EC00071=798156,1112951
EC00072=798156,1112951
EC00073=798156,1112951
EC00074=798156,1112951
EC00075=798156,1112951
EC00076=798156,1112951
EC00077=798156,1112951
EC00078=798156,1112951
EC00079=798156,1112951
EC00080=798156,1112951
EC00081=798156,1112951
EC00082=798156,1112951
EC00083=798156,1112951
EC00084=798156,1112951
EC00085=798156,1112951
EC00086=798156,1112951
EC00087=798156,1112951
EC00088=798156,1112951
EC00089=798156,1112951
EC00090=798156,1112951
EC00091=798156,1112951
EC00092=798156,1112951
EC00093=798156,1112951
EC00094=798156,1112951
EC00095=798156,1112951
EC00096=798156,1112951
EC00097=798156,1112951
EC00098=798156,1112951
EC00099=798156,1112951
EC00100=798156,1112951
EC00101=798156,1112951
EC00102=798156,1112951
EC00103=798156,1112951
EC00104=798156,1112951
EC00105=798156,1112951
EC00106=798156,1112951
EC00107=798156,1112951
EC00108=798156,1112951
EC00109=798156,1112951
EC00110=798156,1112951
EC00111=798156,1112951
EC00112=798156,1112951
EC00113=798156,1112951
EC00114=798156,1112951
EC00115=798156,1112951
EC00116=798156,1112951
EC00117=798156,1112951
EC00118=798156,1112951
EC00119=798156,1112951
EC00120=798156,1112951
EC00121=798156,1112951
EC00122=798156,1112951
EC00123=798156,1112951
EC00124=798156,1112951
EC00125=798156,1112951
EC00126=798156,1112951
EC00127=798156,1112951
EC00128=798156,1112951
EC00129=798156,1112951
EC00130=798156,1112951
EC00131=798156,1112951
EC00132=798156,1112951
EC00133=798156,1112951
EC00134=798156,1112951
EC00135=798156,1112951
EC00136=798156,1112951
EC00137=798156,1112951
EC00138=798156,1112951
EC00139=798156,1112951
EC00140=798156,1112951
EC00141=798156,1112951
EC00142=798156,1112951
EC00143=798156,1112951
EC00144=798156,1112951
EC00145=798156,1112951
EC00146=798156,1112951
EC00147=798156,1112951
EC00148=798156,1112951
EC00149=798156,1112951
EC00150=798156,1112951
EC00151=798156,1112951
EC00152=798156,1112951
EC00153=798156,1112951
EC00154=798156,1112951
EC00155=798156,1112951
EC00156=798156,1112951
EC00157=798156,1112951
EC00158=798156,1112951
EC00159=798156,1112951
EC00160=798156,1112951
EC00161=798156,1112951
EC00162=798156,1112951
EC00163=798156,1112951
EC00164=798156,1112951
EC00165=798156,1112951
EC00166=798156,1112951
EC00167=798156,1112951
EC00168=798156,1112951
EC00169=798156,1112951
EC00170=798156,1112951
EC00171=798156,1112951
EC00172=798156,1112951
EC00173=798156,1112951
EC00174=798156,1112951
EC00175=798156,1112951
EC00176=798156,1112951
EC00177=798156,1112951
EC00178=798156,1112951
EC00179=798156,1112951
EC00180=798156,1112951
EC00181=798156,1112951
EC00182=798156,1112951
EC00183=798156,1112951
EC00184=798156,1112951
EC00185=798156,1112951
EC00186=798156,1112951
EC00187=798156,1112951
EC00188=798155,1112950
EC00189=798156,1112951
EC00190=798156,1112951
EC00191=798156,1112951
EC00192=798156,1112951
EC00193=798156,1112951
EC00194=798156,1112951
EC00195=798156,1112951
EC00196=798156,1112951
EC00197=798156,1112951
EC00198=798156,1112951
EC00199=798156,1112951
EC00200=798156,1112951
EC00201=798156,1112951
EC00202=798156,1112951
EC00203=798156,1112951
EC00204=798156,1112951
EC00205=798156,1112951
EC00206=798156,1112951
EC00207=798156,1112951
EC00208=798156,1112951
EC00209=798156,1112951
EC00210=798156,1112951
EC00211=798156,1112951
EC00212=798156,1112951
EC00213=798156,1112951
EC00214=798156,1112951
EC00215=798156,1112951
EC00216=798156,1112951
EC00217=798156,1112951
EC00218=798156,1112951
EC00219=798156,1112951
EC00220=798156,1112951
EC00221=798156,1112951
EC00222=798156,1112951
EC00223=798156,1112951
EC00224=798156,1112951
EC00225=798156,1112951
EC00226=798156,1112951
EC00227=798156,1112951
EC00228=798156,1112951
EC00229=798156,1112951
EC00230=798156,1112951
EC00231=798156,1112951
EC00232=798156,1112951
EC00233=798156,1112951
EC00234=798156,1112951
EC00235=798156,1112951
EC00236=798156,1112951
EC00237=798156,1112951
EC00238=798156,1112951
EC00239=798156,1112951
EC00240=798156,1112951
EC00241=798156,1112951
EC00242=798156,1112951
EC00243=798156,1112951
EC00244=798156,1112951
EC00245=798156,1112951
EC00246=798156,1112951
EC00247=798156,1112951
EC00248=798156,1112951
EC00249=798156,1112951
EC00250=798156,1112951
EC00251=798156,1112951
EC00252=798156,1112951
EC00253=798156,1112951
EC00254=798156,1112951
EC00255=798156,1112951
EC00256=798156,1112951
EC00257=798156,1112951
EC00258=798156,1112951
EC00259=798156,1112951
EC00260=798156,1112951
EC00261=798156,1112951
EC00262=798156,1112951
EC00263=798156,1112951
EC00264=798156,1112951
EC00265=798156,1112951
EC00266=798156,1112951
EC00267=798156,1112951
EC00268=798156,1112951
EC00269=798156,1112951
EC00270=798156,1112951
EC00271=798156,1112951
EC00272=798156,1112951
EC00273=798156,1112951
EC00274=798156,1112951
EC00275=798156,1112951
EC00276=798156,1112951
EC00277=798156,1112951
EC00278=798156,1112951
EC00279=798156,1112951
EC00280=798156,1112951
EC00281=798155,1112951
EC00282=798156,1112951
EC00283=798156,1112951
EC00284=798156,1112951
EC00285=798156,1112951
EC00286=798156,1112951
EC00287=798156,1112951
EC00288=798156,1112951
EC00289=798156,1112951
EC00290=798156,1112951
EC00291=798156,1112951
EC00292=798156,1112951
EC00293=798156,1112951
EC00294=798156,1112951
EC00295=798156,1112951
EC00296=798156,1112951
EC00297=798156,1112951
EC00298=798156,1112951
EC00299=798156,1112951
EC00300=798156,1112951
EC00301=798156,1112951
EC00302=798156,1112951
EC00303=798156,1112951
EC00304=798156,1112951
EC00305=798156,1112951
EC00306=798156,1112951
EC00307=798156,1112951
EC00308=798156,1112951
EC00309=798156,1112951
EC00310=798156,1112951
EC00311=798156,1112951
EC00312=798156,1112951
EC00313=798156,1112951
EC00314=798156,1112951
EC00315=798156,1112951
EC00316=798156,1112951
EC00317=798156,1112951
EC00318=798156,1112951
EC00319=798156,1112951
EC00320=798156,1112951
EC00321=798156,1112951
EC00322=798156,1112951
EC00323=798156,1112951
EC00324=798156,1112951
EC00325=798156,1112951
EC00326=798156,1112951
EC00327=798156,1112951
EC00328=798156,1112951
EC00329=798156,1112951
EC00330=798156,1112951
EC00331=798156,1112951
EC00332=798156,1112951
EC00333=798156,1112951
EC00334=798156,1112951
EC00335=798156,1112951
EC00336=798156,1112951
EC00337=798156,1112951
EC00338=798156,1112951
EC00339=798156,1112951
EC00340=798156,1112951
EC00341=798156,1112951
EC00342=798156,1112951
EC00343=798156,1112951
EC00344=798156,1112951
EC00345=798156,1112951
EC00346=798156,1112951
EC00347=798156,1112951
EC00348=798156,1112951
EC00349=798156,1112951
EC00350=798156,1112951
EC00351=798156,1112951
EC00352=798156,1112951
EC00353=798156,1112951
EC00354=798156,1112951
EC00355=798156,1112951
EC00356=798156,1112951
EC00357=798156,1112951
EC00358=798156,1112951
EC00359=798156,1112951
EC00360=798156,1112951
EC00361=798156,1112951
EC00362=798155,1112950
EC00363=798156,1112951
EC00364=798156,1112951
EC00365=798156,1112951
EC00366=798156,1112951
EC00367=798156,1112951
EC00368=798156,1112951
EC00369=798155,1112951
EC00370=798155,1112951
EC00371=798156,1112951
EC00372=798156,1112951
EC00373=798156,1112951
EC00374=798156,1112951
EC00375=798156,1112951
EC00376=798156,1112951
EC00377=798156,1112951
EC00378=798156,1112951
EC00379=798155,1112950
EC00380=798156,1112951
EC00381=798156,1112951
EC00382=798156,1112951
EC00383=798156,1112951
EC00384=798156,1112951
EC00385=798156,1112951
EC00386=798156,1112951
EC00387=798156,1112951
EC00388=798156,1112951
EC00389=798156,1112951
EC00390=798156,1112951
EC00391=798156,1112951
EC00392=798156,1112951
EC00393=798156,1112951
EC00394=798156,1112951
EC00395=798156,1112951
EC00396=798156,1112951
EC00397=798156,1112951
EC00398=798156,1112951
EC00399=798156,1112951
EC00400=798156,1112951
EC00401=798156,1112951
EC00402=798156,1112951
EC00403=798156,1112951
EC00404=798156,1112951
EC00405=798156,1112951
EC00406=798156,1112951
EC00407=798155,1112950
EC00408=798156,1112951
EC00409=798156,1112951
EC00410=798156,1112951
EC00411=798156,1112951
EC00412=798156,1112951
EC00413=798156,1112951
EC00414=798156,1112951
EC00415=798156,1112951
EC00416=798156,1112951
EC00417=798156,1112951
EC00418=798156,1112951
EC00419=798156,1112951
EC00420=798156,1112951
EC00421=798156,1112951
EC00422=798156,1112951
EC00423=798156,1112951
EC00424=798156,1112951
EC00425=798156,1112951
EC00426=798156,1112951
EC00427=798156,1112951
EC00428=798156,1112951
EC00429=798156,1112951
EC00430=798156,1112951
EC00431=798156,1112951
EC00432=798156,1112951
EC00433=798156,1112951
EC00434=798156,1112951
EC00435=798156,1112951
EC00436=798156,1112951
EC00437=798156,1112951
EC00438=798156,1112951
EC00439=798156,1112951
EC00440=798156,1112951
EC00441=798156,1112951
EC00442=798155,1112950
EC00443=798156,1112951
EC00444=798156,1112951
EC00445=798156,1112951
EC00446=798156,1112951
EC00447=798156,1112951
EC00448=798156,1112951
EC00449=798156,1112951
EC00450=798156,1112951
EC00451=798156,1112951
EC00452=798156,1112951
EC00453=798156,1112951
EC00454=798156,1112951
EC00455=798156,1112951
EC00456=798156,1112951
EC00457=798156,1112951
EC00458=798156,1112951
EC00459=798156,1112951
EC00460=798156,1112951
EC00461=798156,1112951
EC00462=798156,1112951
EC00463=798156,1112951
EC00464=798156,1112951
EC00465=798156,1112951
EC00466=798156,1112951
EC00467=798156,1112951
EC00468=798156,1112951
EC00469=798156,1112951
EC00470=798156,1112951
EC00471=798156,1112951
EC00472=798156,1112951
EC00473=798156,1112951
EC00474=798156,1112951
EC00475=798156,1112951
EC00476=798156,1112951
EC00477=798156,1112951
EC00478=798156,1112951
EC00479=798156,1112951
EC00480=798156,1112951
EC00481=798156,1112951
EC00482=798156,1112951
EC00483=798156,1112951
EC00484=798156,1112951
EC00485=798156,1112951
EC00486=798156,1112951
EC00487=798156,1112951
EC00488=798156,1112951
EC00489=798156,1112951
EC00490=798156,1112951
EC00491=798156,1112951
EC00492=798156,1112951
EC00493=798156,1112951
EC00494=798156,1112951
EC00495=798156,1112951
EC00496=798156,1112951
EC00497=798156,1112951
EC00498=798156,1112951
EC00499=798156,1112951
EC00500=798156,1112951
EC00501=798156,1112951
EC00502=798156,1112951
EC00503=798156,1112951
EC00504=798156,1112951
EC00505=798156,1112951
EC00506=798156,1112951
EC00507=798156,1112951
EC00508=798156,1112951
EC00509=798156,1112951
EC00510=798156,1112951
EC00511=798156,1112951
EC00512=798156,1112951
EC00513=798156,1112951
EC00514=798156,1112951
EC00515=798156,1112951
EC00516=798156,1112951
EC00517=798156,1112951
EC00518=798156,1112951
EC00519=798156,1112951
EC00520=798156,1112951
EC00521=798156,1112951
EC00522=798156,1112951
EC00523=798156,1112951
EC00524=798156,1112951
EC00525=798156,1112951
EC00526=798156,1112951
EC00527=798156,1112951
EC00528=798156,1112951
EC00529=798156,1112951
EC00530=798156,1112951
EC00531=798156,1112951
EC00532=798156,1112951
EC00533=798156,1112951
EC00534=798156,1112951
EC00535=798156,1112951
EC00536=798156,1112951
EC00537=798156,1112951
EC00538=798156,1112951
EC00539=798156,1112951
EC00540=798156,1112951
EC00541=798156,1112951
EC00542=798156,1112951
EC00543=798156,1112951
EC00544=798156,1112951
EC00545=798156,1112951
EC00546=798156,1112951
EC00547=798156,1112951
EC00548=798156,1112951
EC00549=798156,1112951
EC00550=798156,1112951
EC00551=798156,1112951
EC00552=798156,1112951
EC00553=798156,1112951
EC00554=798156,1112951
EC00555=798156,1112951
EC00556=798156,1112951
EC00557=798156,1112951
EC00558=798156,1112951
EC00559=798156,1112951
EC00560=798156,1112951
EC00561=798156,1112951
EC00562=798156,1112951
EC00563=798156,1112951
EC00564=798156,1112951
EC00565=798156,1112951
EC00566=798156,1112951
EC00567=798156,1112951
EC00568=798156,1112951
EC00569=798156,1112951
EC00570=798156,1112951
EC00571=798156,1112951
EC00572=798156,1112951
EC00573=798156,1112951
EC00574=798156,1112951
EC00575=798156,1112951
EC00576=798156,1112951
EC00577=798156,1112951
EC00578=798156,1112951
EC00579=798156,1112951
EC00580=798156,1112951
EC00581=798156,1112951
EC00582=798156,1112951
EC00583=798156,1112951
EC00584=798156,1112951
EC00585=798156,1112951
EC00586=798156,1112951
EC00587=798156,1112951
EC00588=798156,1112951
EC00589=798156,1112951
EC00590=798156,1112951
EC00591=798156,1112951
EC00592=798156,1112951
EC00593=798156,1112951
EC00594=798156,1112951
EC00595=798156,1112951
EC00596=798156,1112951
EC00597=798156,1112951
EC00598=798156,1112951
EC00599=798156,1112951
EC00600=798156,1112951
EC00601=798156,1112951
EC00602=798156,1112951
EC00603=798156,1112951
EC00604=798156,1112951
EC00605=798156,1112951
EC00606=798156,1112951
EC00607=798156,1112951
EC00608=798156,1112951
EC00609=798156,1112951
EC00610=798156,1112951
EC00611=798156,1112951
EC00612=798156,1112951
EC00613=798156,1112951
EC00614=798156,1112951
EC00615=798156,1112951
EC00616=798156,1112951
EC00617=798156,1112951
EC00618=798156,1112951
EC00619=798156,1112951
EC00620=798156,1112951
EC00621=798156,1112951
EC00622=798156,1112951
EC00623=798156,1112951
EC00624=798156,1112951
EC00625=798156,1112951
EC00626=798156,1112951
EC00627=798156,1112951
EC00628=798156,1112951
EC00629=798156,1112951
EC00630=798156,1112951
EC00631=798155,1112950
EC00632=798156,1112951
EC00633=798156,1112951
EC00634=798156,1112951
EC00635=798156,1112951
EC00636=798156,1112951
EC00637=798156,1112951
EC00638=798156,1112951
EC00639=798156,1112951
EC00640=798156,1112951
EC00641=798156,1112951
EC00642=798156,1112951
EC00643=798156,1112951
EC00644=798156,1112951
EC00645=798156,1112951
EC00646=798156,1112951
EC00647=798156,1112951
EC00648=798156,1112951
EC00649=798156,1112951
EC00650=798156,1112951
EC00651=798156,1112951
EC00652=798156,1112951
EC00653=798156,1112951
EC00654=798156,1112951
EC00655=798156,1112951
EC00656=798156,1112951
EC00657=798156,1112951
EC00658=798156,1112951
EC00659=798156,1112951
EC00660=798156,1112951
EC00661=798156,1112951
EC00662=798156,1112951
EC00663=798156,1112951
EC00664=798156,1112951
EC00665=798156,1112951
EC00666=798156,1112951
EC00667=798156,1112951
EC00668=798156,1112951
EC00669=798156,1112951
EC00670=798156,1112951
EC00671=798156,1112951
EC00672=798156,1112951
EC00673=798156,1112951
EC00674=798156,1112951
EC00675=798156,1112951
EC00676=798156,1112951
EC00677=798156,1112951
EC00678=798156,1112951
EC00679=798156,1112951
EC00680=798156,1112951
EC00681=798156,1112951
EC00682=798156,1112951
EC00683=798156,1112951
EC00684=798156,1112951
EC00685=798156,1112951
EC00686=798156,1112951
EC00687=798156,1112951
EC00688=798156,1112951
EC00689=798156,1112951
EC00690=798156,1112951
EC00691=798156,1112951
EC00692=798156,1112951
EC00693=798156,1112951
EC00694=798156,1112951
EC00695=798156,1112951
EC00696=798156,1112951
EC00697=798156,1112951
EC00698=798156,1112951
EC00699=798156,1112951
EC00700=798156,1112951
EC00701=798156,1112951
EC00702=798156,1112951
EC00703=798156,1112951
EC00704=798156,1112951
EC00705=798156,1112951
EC00706=798156,1112951
EC00707=798156,1112951
EC00708=798156,1112951
EC00709=798156,1112951
EC00710=798156,1112951
EC00711=798156,1112951
EC00712=798156,1112951
EC00713=798156,1112951
EC00714=798156,1112951
EC00715=798156,1112951
EC00716=798156,1112951
EC00717=798156,1112951
EC00718=798156,1112951
EC00719=798156,1112951
EC00720=798156,1112951
EC00721=798156,1112951
EC00722=798156,1112951
EC00723=798156,1112951
EC00724=798156,1112951
EC00725=798156,1112951
EC00726=798156,1112951
EC00727=798156,1112951
EC00728=798156,1112951
EC00729=798156,1112951
EC00730=798156,1112951
EC00731=798156,1112951
EC00732=798156,1112951
EC00733=798156,1112951
EC00734=798156,1112951
EC00735=798156,1112951
EC00736=798156,1112951
EC00737=798156,1112951
EC00738=798156,1112951
EC00739=798156,1112951
EC00740=798156,1112951
EC00741=798156,1112951
EC00742=798156,1112951
EC00743=798156,1112951
EC00744=798156,1112951
EC00745=798156,1112951
EC00746=798156,1112951
EC00747=798156,1112951
EC00748=798156,1112951
EC00749=798156,1112951
EC00750=798155,1112951
EC00751=798155,1112951
EC00752=798156,1112951
EC00753=798156,1112951
EC00754=798156,1112951
EC00755=798156,1112951
EC00756=798156,1112951
EC00757=798156,1112951
EC00758=798156,1112951
EC00759=798156,1112951
EC00760=798155,1112950
EC00761=798155,1112950
EC00762=798155,1112950
EC00763=798155,1112950
EC00764=798155,1112950
EC00765=798156,1112951
EC00766=798156,1112951
EC00767=798156,1112951
EC00768=798156,1112951
EC00769=798156,1112951
EC00770=798156,1112951
EC00771=798156,1112951
EC00772=798156,1112951
EC00773=798156,1112951
EC00774=798156,1112951
EC00775=798156,1112951
EC00776=798156,1112951
EC00777=798156,1112951
EC00778=798156,1112951
EC00779=798156,1112951
EC00780=798156,1112951
EC00781=798156,1112951
EC00782=798156,1112951
EC00783=798156,1112951
EC00784=798156,1112951
EC00785=798156,1112951
EC00786=798156,1112951
EC00787=798156,1112951
EC00788=798156,1112951
EC00789=798156,1112951
EC00790=798156,1112951
EC00791=798156,1112951
EC00792=798156,1112951
EC00793=798156,1112951
EC00794=798156,1112951
EC00795=798156,1112951
EC00796=798156,1112951
EC00797=798156,1112951
EC00798=798156,1112951
EC00799=798156,1112951
EC00800=798156,1112951
EC00801=798156,1112951
EC00802=798156,1112951
EC00803=798156,1112951
EC00804=798156,1112951
EC00805=798156,1112951
EC00806=798156,1112951
EC00807=798156,1112951
EC00808=798156,1112951
EC00809=798156,1112951
EC00810=798156,1112951
EC00811=798156,1112951
EC00812=798156,1112951
EC00813=798156,1112951
EC00814=798156,1112951
EC00815=798156,1112951
EC00816=798156,1112951
EC00817=798156,1112951
EC00818=798156,1112951
EC00819=798156,1112951
EC00820=798156,1112951
EC00821=798156,1112951
EC00822=798156,1112951
EC00823=798156,1112951
EC00824=798156,1112951
EC00825=798156,1112951
EC00826=798156,1112951
EC00827=798156,1112951
EC00828=798156,1112951
EC00829=798156,1112951
EC00830=798156,1112951
EC00831=798156,1112951
EC00832=798156,1112951
EC00833=798156,1112951
EC00834=798156,1112951
EC00835=798156,1112951
EC00836=798156,1112951
EC00837=798156,1112951
EC00838=798156,1112951
EC00839=798156,1112951
EC00840=798156,1112951
EC00841=798156,1112951
EC00842=798156,1112951
